C03645=1217.318,-29.503,-40.529,-179.892,5.418,148.913
C03646=1217.324,-29.753,-40.516,-179.895,5.418,148.914
C03647=1217.328,-30.003,-40.503,-179.897,5.418,148.915
C03648=1217.333,-30.252,-40.490,-179.899,5.417,148.915
C03649=1217.339,-30.503,-40.476,-179.902,5.417,148.916
C03650=1217.344,-30.752,-40.464,-179.904,5.417,148.917
C03651=1217.349,-31.001,-40.451,-179.907,5.417,148.918
C03652=1217.354,-31.252,-40.438,-179.909,5.416,148.918
C03653=1217.359,-31.501,-40.425,-179.912,5.417,148.919
C03654=1217.364,-31.750,-40.413,-179.914,5.416,148.920
C03655=1217.369,-32.000,-40.398,-179.917,5.416,148.920
C03656=1217.374,-32.249,-40.386,-179.919,5.416,148.921
C03657=1217.380,-32.499,-40.373,-179.922,5.415,148.922
C03658=1217.384,-32.749,-40.360,-179.924,5.415,148.922
C03659=1217.390,-32.998,-40.347,-179.926,5.415,148.923
C03660=1217.395,-33.248,-40.334,-179.928,5.414,148.924
C03661=1217.400,-33.498,-40.321,-179.931,5.414,148.924
C03662=1217.405,-33.747,-40.308,-179.933,5.414,148.925
C03663=1217.411,-33.997,-40.296,-179.936,5.414,148.926
C03664=1217.415,-34.247,-40.283,-179.939,5.413,148.926
C03665=1217.420,-34.496,-40.270,-179.941,5.414,148.927
C03666=1217.425,-34.745,-40.257,-179.943,5.413,148.928
C03667=1217.431,-34.996,-40.244,-179.946,5.413,148.928
C03668=1217.436,-35.245,-40.231,-179.948,5.413,148.929
C03669=1217.441,-35.494,-40.219,-179.951,5.412,148.930
C03670=1217.446,-35.743,-40.206,-179.953,5.412,148.931
C03671=1217.451,-35.994,-40.192,-179.955,5.412,148.931
C03672=1217.457,-36.244,-40.181,-179.958,5.412,148.932
C03673=1217.462,-36.493,-40.168,-179.961,5.411,148.933
C03674=1217.466,-36.743,-40.155,-179.963,5.412,148.933
C03675=1217.471,-36.992,-40.142,-179.966,5.411,148.934
C03676=1217.477,-37.242,-40.129,-179.968,5.411,148.935
C03677=1217.482,-37.491,-40.117,-179.970,5.411,148.935
C03678=1217.487,-37.741,-40.104,-179.973,5.411,148.936
C03679=1217.492,-37.991,-40.091,-179.975,5.411,148.937
C03680=1217.497,-38.240,-40.078,-179.978,5.410,148.938
C03681=1217.502,-38.489,-40.066,-179.980,5.410,148.938
C03682=1217.508,-38.740,-40.053,-179.982,5.410,148.939
C03683=1217.513,-38.990,-40.040,-179.985,5.409,148.939
C03684=1217.518,-39.239,-40.028,-179.987,5.409,148.940
C03685=1217.523,-39.488,-40.015,-179.989,5.409,148.941
C03686=1217.528,-39.738,-40.002,-179.992,5.409,148.942
C03687=1217.533,-39.988,-39.990,-179.995,5.408,148.942
C03688=1217.538,-40.238,-39.978,-179.997,5.409,148.943
C03689=1217.543,-40.487,-39.965,-179.999,5.408,148.944
C03690=1217.549,-40.737,-39.952,179.998,5.408,148.944
C03691=1217.554,-40.986,-39.939,179.996,5.408,148.945
C03692=1217.559,-41.236,-39.926,179.993,5.408,148.946
C03693=1217.564,-41.486,-39.914,179.991,5.407,148.946
C03694=1217.570,-41.735,-39.902,179.988,5.407,148.947
C03695=1217.574,-41.985,-39.889,179.986,5.407,148.948
C03696=1217.579,-42.234,-39.876,179.984,5.407,148.949
C03697=1217.585,-42.484,-39.864,179.981,5.407,148.949
C03698=1217.590,-42.734,-39.852,179.978,5.406,148.950
C03699=1217.595,-42.983,-39.839,179.976,5.407,148.951
C03700=1217.599,-43.233,-39.826,179.974,5.406,148.951
C03701=1217.605,-43.483,-39.814,179.971,5.406,148.952
C03702=1217.610,-43.732,-39.802,179.969,5.406,148.953
C03703=1217.615,-43.982,-39.789,179.967,5.405,148.953
C03704=1217.620,-44.231,-39.777,179.964,5.405,148.954
C03705=1217.625,-44.482,-39.764,179.962,5.405,148.955
C03706=1217.630,-44.731,-39.752,179.959,5.405,148.955
C03707=1217.635,-44.980,-39.739,179.957,5.405,148.956
C03708=1217.641,-45.230,-39.727,179.955,5.404,148.957
C03709=1217.646,-45.479,-39.715,179.952,5.404,148.957
C03710=1217.651,-45.729,-39.702,179.950,5.404,148.958
C03711=1217.656,-45.979,-39.690,179.947,5.404,148.959
C03712=1217.661,-46.229,-39.677,179.944,5.403,148.960
C03713=1217.666,-46.478,-39.665,179.942,5.404,148.960
C03714=1217.671,-46.728,-39.653,179.940,5.403,148.961
C03715=1217.677,-46.977,-39.640,179.938,5.404,148.962
C03716=1217.682,-47.227,-39.628,179.935,5.403,148.962
C03717=1217.687,-47.476,-39.616,179.932,5.403,148.963
C03718=1217.692,-47.726,-39.603,179.930,5.403,148.964
C03719=1217.697,-47.976,-39.591,179.928,5.402,148.964
C03720=1217.702,-48.226,-39.578,179.925,5.402,148.965
C03721=1217.708,-48.495,-39.566,179.923,5.402,148.966
C03722=1217.714,-48.765,-39.551,179.920,5.402,148.967
C03723=1217.719,-49.036,-39.538,179.917,5.401,148.967
C03724=1217.725,-49.305,-39.525,179.915,5.401,148.968
C03725=1217.730,-49.555,-39.513,179.913,5.401,148.969
C03726=1217.735,-49.805,-39.500,179.910,5.401,148.969
C03727=1217.740,-50.055,-39.488,179.908,5.401,148.970
C03728=1217.745,-50.304,-39.476,179.905,5.401,148.971
C03729=1217.751,-50.554,-39.464,179.903,5.400,148.971
C03730=1217.756,-50.803,-39.451,179.901,5.400,148.972
C03731=1217.760,-51.053,-39.440,179.898,5.400,148.973
C03732=1217.766,-51.302,-39.427,179.896,5.400,148.974
C03733=1217.771,-51.552,-39.415,179.893,5.400,148.974
C03734=1217.776,-51.801,-39.403,179.890,5.399,148.975
C03735=1217.782,-52.051,-39.391,179.888,5.400,148.976
C03736=1217.787,-52.301,-39.378,179.886,5.399,148.976
C03737=1217.792,-52.551,-39.366,179.883,5.399,148.977
C03738=1217.798,-52.801,-39.355,179.881,5.399,148.978
C03739=1217.801,-53.050,-39.342,179.878,5.399,148.979
C03740=1217.807,-53.300,-39.330,179.876,5.399,148.979
C03741=1217.812,-53.550,-39.318,179.874,5.399,148.980
C03742=1217.817,-53.800,-39.306,179.871,5.398,148.980
C03743=1217.822,-54.049,-39.293,179.869,5.398,148.981
C03744=1217.827,-54.298,-39.282,179.867,5.398,148.982
C03745=1217.833,-54.548,-39.270,179.865,5.398,148.982
C03746=1217.838,-54.798,-39.257,179.862,5.397,148.983
C03747=1217.843,-55.048,-39.245,179.859,5.397,148.984
C03748=1217.848,-55.297,-39.233,179.857,5.397,148.985
C03749=1217.853,-55.547,-39.222,179.854,5.397,148.985
C03750=1217.858,-55.797,-39.210,179.852,5.397,148.986
C03751=1217.863,-56.046,-39.197,179.850,5.397,148.987
C03752=1217.869,-56.296,-39.185,179.847,5.396,148.987
C03753=1217.874,-56.546,-39.173,179.845,5.397,148.988
C03754=1217.879,-56.795,-39.161,179.842,5.396,148.989
C03755=1217.884,-57.045,-39.149,179.840,5.397,148.990
C03756=1217.890,-57.295,-39.138,179.837,5.396,148.990
C03757=1217.895,-57.544,-39.125,179.835,5.396,148.991
C03758=1217.899,-57.794,-39.114,179.833,5.396,148.992
C03759=1217.905,-58.043,-39.102,179.830,5.395,148.992
C03760=1217.910,-58.293,-39.089,179.828,5.395,148.993
C03761=1217.915,-58.542,-39.078,179.826,5.395,148.994
C03762=1217.920,-58.792,-39.066,179.824,5.395,148.994
C03763=1217.926,-59.042,-39.054,179.821,5.395,148.995
C03764=1217.931,-59.292,-39.042,179.818,5.394,148.996
C03765=1217.935,-59.541,-39.030,179.816,5.395,148.996
C03766=1217.941,-59.791,-39.018,179.814,5.394,148.997
C03767=1217.946,-60.040,-39.006,179.812,5.395,148.998
C03768=1217.951,-60.290,-38.994,179.809,5.394,148.998
C03769=1217.956,-60.540,-38.983,179.806,5.394,148.999
C03770=1217.961,-60.790,-38.971,179.804,5.394,149.000
C03771=1217.966,-61.040,-38.959,179.801,5.394,149.001
C03772=1217.971,-61.289,-38.947,179.799,5.394,149.001
C03773=1217.977,-61.539,-38.935,179.797,5.393,149.002
C03774=1217.982,-61.788,-38.924,179.795,5.394,149.003
C03775=1217.987,-62.038,-38.912,179.792,5.393,149.003
C03776=1217.993,-62.288,-38.900,179.790,5.393,149.004
C03777=1217.997,-62.537,-38.888,179.788,5.393,149.005
C03778=1218.003,-62.787,-38.876,179.785,5.392,149.005
C03779=1218.008,-63.037,-38.864,179.783,5.393,149.006
C03780=1218.013,-63.286,-38.853,179.780,5.392,149.007
C03781=1218.018,-63.536,-38.841,179.778,5.392,149.007
C03782=1218.024,-63.786,-38.829,179.776,5.392,149.008
C03783=1218.028,-64.036,-38.818,179.773,5.392,149.009
C03784=1218.033,-64.285,-38.806,179.771,5.392,149.010
C03785=1218.038,-64.535,-38.794,179.768,5.392,149.010
C03786=1218.044,-64.784,-38.783,179.766,5.392,149.011
C03787=1218.050,-65.034,-38.771,179.763,5.391,149.012
C03788=1218.054,-65.283,-38.760,179.761,5.391,149.012
C03789=1218.060,-65.533,-38.748,179.759,5.391,149.013
C03790=1218.064,-65.783,-38.736,179.756,5.391,149.014
C03791=1218.070,-66.033,-38.724,179.754,5.391,149.014
C03792=1218.075,-66.283,-38.713,179.752,5.390,149.015
C03793=1218.080,-66.532,-38.701,179.750,5.391,149.016
C03794=1218.086,-66.782,-38.690,179.747,5.390,149.016
C03795=1218.091,-67.031,-38.678,179.744,5.390,149.017
C03796=1218.096,-67.281,-38.667,179.742,5.390,149.018
C03797=1218.101,-67.531,-38.655,179.739,5.390,149.018
C03798=1218.106,-67.780,-38.643,179.737,5.390,149.019
C03799=1218.111,-68.030,-38.631,179.735,5.390,149.020
C03800=1218.116,-68.280,-38.620,179.733,5.390,149.021
C03801=1218.122,-68.529,-38.608,179.730,5.390,149.021
C03802=1218.127,-68.779,-38.597,179.728,5.390,149.022
C03803=1218.132,-69.029,-38.585,179.725,5.389,149.023
C03804=1218.137,-69.279,-38.574,179.723,5.389,149.023
C03805=1218.143,-69.529,-38.562,179.720,5.389,149.024
C03806=1218.147,-69.778,-38.551,179.718,5.389,149.025
C03807=1218.153,-70.028,-38.540,179.716,5.389,149.025
C03808=1218.158,-70.277,-38.528,179.714,5.388,149.026
C03809=1218.163,-70.527,-38.516,179.711,5.389,149.027
C03810=1218.168,-70.777,-38.505,179.709,5.388,149.027
C03811=1218.174,-71.027,-38.493,179.706,5.388,149.028
C03812=1218.179,-71.276,-38.482,179.704,5.388,149.029
C03813=1218.184,-71.526,-38.470,179.701,5.388,149.030
C03814=1218.189,-71.775,-38.459,179.699,5.388,149.030
C03815=1218.194,-72.025,-38.448,179.697,5.388,149.031
C03816=1218.199,-72.275,-38.436,179.694,5.388,149.032
C03817=1218.204,-72.524,-38.425,179.692,5.388,149.032
C03818=1218.210,-72.774,-38.414,179.690,5.388,149.033
C03819=1218.215,-73.024,-38.403,179.688,5.387,149.034
C03820=1218.220,-73.274,-38.391,179.685,5.387,149.034
C03821=1218.226,-73.523,-38.380,179.683,5.387,149.035
C03822=1218.231,-73.773,-38.368,179.680,5.387,149.036
C03823=1218.236,-74.022,-38.357,179.678,5.387,149.036
C03824=1218.240,-74.272,-38.345,179.675,5.386,149.037
C03825=1218.247,-74.542,-38.333,179.673,5.387,149.038
C03826=1218.252,-74.813,-38.321,179.671,5.386,149.039
C03827=1218.258,-75.084,-38.309,179.667,5.386,149.039
C03828=1218.264,-75.354,-38.296,179.665,5.387,149.040
C03829=1218.268,-75.603,-38.285,179.663,5.386,149.041
C03830=1218.274,-75.854,-38.274,179.660,5.386,149.042
C03831=1218.279,-76.103,-38.263,179.658,5.386,149.042
C03832=1218.284,-76.353,-38.252,179.656,5.385,149.043
C03833=1218.290,-76.603,-38.240,179.654,5.386,149.044
C03834=1218.295,-76.853,-38.229,179.651,5.385,149.044
C03835=1218.301,-77.102,-38.218,179.649,5.386,149.045
C03836=1218.305,-77.352,-38.206,179.646,5.385,149.046
C03837=1218.310,-77.601,-38.195,179.644,5.385,149.046
C03838=1218.316,-77.852,-38.184,179.641,5.385,149.047
C03839=1218.321,-78.101,-38.173,179.639,5.385,149.048
C03840=1218.326,-78.350,-38.162,179.637,5.385,149.048
C03841=1218.331,-78.600,-38.150,179.635,5.385,149.049
C03842=1218.337,-78.850,-38.140,179.632,5.384,149.050
C03843=1218.341,-79.099,-38.128,179.630,5.384,149.050
C03844=1218.346,-79.349,-38.117,179.628,5.384,149.051
C03845=1218.352,-79.599,-38.106,179.625,5.384,149.052
C03846=1218.357,-79.849,-38.095,179.623,5.384,149.052
C03847=1218.362,-80.098,-38.084,179.620,5.384,149.053
C03848=1218.368,-80.349,-38.072,179.618,5.384,149.054
C03849=1218.373,-80.598,-38.062,179.615,5.384,149.055
C03850=1218.378,-80.847,-38.050,179.613,5.384,149.055
C03851=1218.383,-81.098,-38.039,179.611,5.384,149.056
C03852=1218.389,-81.347,-38.028,179.609,5.384,149.057
C03853=1218.393,-81.596,-38.017,179.606,5.383,149.057
C03854=1218.398,-81.847,-38.006,179.604,5.384,149.058
C03855=1218.404,-82.096,-37.995,179.602,5.383,149.059
C03856=1218.409,-82.345,-37.983,179.600,5.383,149.059
C03857=1218.414,-82.596,-37.973,179.597,5.383,149.060
C03858=1218.419,-82.845,-37.962,179.594,5.383,149.061
C03859=1218.425,-83.095,-37.951,179.592,5.383,149.061
C03860=1218.430,-83.344,-37.940,179.589,5.382,149.062
C03861=1218.435,-83.594,-37.929,179.587,5.383,149.063
C03862=1218.440,-83.844,-37.918,179.585,5.382,149.064
C03863=1218.445,-84.093,-37.907,179.583,5.382,149.064
C03864=1218.451,-84.343,-37.896,179.580,5.382,149.065
C03865=1218.456,-84.593,-37.885,179.578,5.382,149.066
C03866=1218.461,-84.843,-37.874,179.576,5.382,149.066
C03867=1218.466,-85.092,-37.863,179.574,5.382,149.067
C03868=1218.471,-85.343,-37.853,179.571,5.382,149.068
C03869=1218.477,-85.592,-37.841,179.569,5.382,149.068
C03870=1218.482,-85.842,-37.830,179.566,5.382,149.069
C03871=1218.487,-86.091,-37.820,179.564,5.382,149.070
C03872=1218.492,-86.341,-37.809,179.562,5.381,149.070
C03873=1218.497,-86.591,-37.798,179.560,5.382,149.071
C03874=1218.503,-86.840,-37.787,179.557,5.381,149.072
C03875=1218.508,-87.090,-37.776,179.555,5.382,149.072
C03876=1218.514,-87.340,-37.765,179.552,5.381,149.073
C03877=1218.518,-87.589,-37.754,179.550,5.381,149.074
C03878=1218.523,-87.840,-37.743,179.548,5.381,149.075
C03879=1218.529,-88.089,-37.733,179.545,5.381,149.075
C03880=1218.534,-88.339,-37.722,179.543,5.381,149.076
C03881=1218.539,-88.588,-37.711,179.540,5.380,149.077
C03882=1218.544,-88.838,-37.700,179.539,5.380,149.077
C03883=1218.550,-89.087,-37.689,179.536,5.380,149.078
C03884=1218.555,-89.338,-37.678,179.534,5.380,149.079
C03885=1218.560,-89.588,-37.668,179.531,5.380,149.079
C03886=1218.565,-89.837,-37.657,179.529,5.380,149.080
C03887=1218.570,-90.087,-37.646,179.526,5.380,149.081
C03888=1218.576,-90.336,-37.635,179.524,5.380,149.081
C03889=1218.581,-90.586,-37.625,179.522,5.380,149.082
C03890=1218.586,-90.836,-37.615,179.520,5.380,149.083
C03891=1218.591,-91.085,-37.603,179.517,5.379,149.083
C03892=1218.596,-91.335,-37.593,179.515,5.380,149.084
C03893=1218.601,-91.585,-37.583,179.513,5.379,149.085
C03894=1218.607,-91.834,-37.571,179.510,5.380,149.085
C03895=1218.612,-92.085,-37.560,179.508,5.379,149.086
C03896=1218.618,-92.333,-37.550,179.506,5.380,149.087
C03897=1218.623,-92.584,-37.539,179.503,5.379,149.088
C03898=1218.628,-92.834,-37.528,179.501,5.379,149.088
C03899=1218.633,-93.083,-37.518,179.499,5.379,149.089
C03900=1218.638,-93.333,-37.507,179.497,5.379,149.089
C03901=1218.644,-93.583,-37.497,179.494,5.379,149.090
C03902=1218.649,-93.833,-37.486,179.492,5.379,149.091
C03903=1218.654,-94.082,-37.475,179.489,5.379,149.092
C03904=1218.659,-94.332,-37.465,179.487,5.379,149.092
C03905=1218.665,-94.582,-37.454,179.484,5.378,149.093
C03906=1218.669,-94.831,-37.443,179.483,5.378,149.094
C03907=1218.675,-95.081,-37.433,179.480,5.378,149.094
C03908=1218.680,-95.330,-37.423,179.478,5.378,149.095
C03909=1218.685,-95.581,-37.412,179.475,5.378,149.096
C03910=1218.691,-95.829,-37.401,179.473,5.378,149.096
C03911=1218.696,-96.080,-37.391,179.471,5.378,149.097
C03912=1218.701,-96.329,-37.380,179.469,5.378,149.098
C03913=1218.706,-96.580,-37.370,179.466,5.378,149.099
C03914=1218.712,-96.829,-37.360,179.464,5.378,149.099
C03915=1218.717,-97.079,-37.348,179.462,5.377,149.100
C03916=1218.722,-97.328,-37.338,179.460,5.378,149.100
C03917=1218.727,-97.578,-37.328,179.457,5.377,149.101
C03918=1218.733,-97.828,-37.317,179.455,5.378,149.102
C03919=1218.738,-98.078,-37.307,179.452,5.377,149.103
C03920=1218.742,-98.327,-37.296,179.450,5.378,149.103
C03921=1218.748,-98.576,-37.286,179.448,5.377,149.104
C03922=1218.753,-98.827,-37.276,179.446,5.377,149.104
C03923=1218.759,-99.076,-37.265,179.443,5.377,149.105
C03924=1218.764,-99.326,-37.255,179.441,5.377,149.106
C03925=1218.769,-99.576,-37.245,179.438,5.377,149.107
C03926=1218.774,-99.826,-37.234,179.436,5.377,149.107
C03927=1218.779,-100.075,-37.223,179.434,5.377,149.108
C03928=1218.785,-100.325,-37.213,179.432,5.377,149.109
C03929=1218.790,-100.596,-37.202,179.429,5.377,149.109
C03930=1218.796,-100.868,-37.190,179.427,5.377,149.110
C03931=1218.801,-101.139,-37.180,179.424,5.377,149.111
C03932=1218.808,-101.410,-37.168,179.421,5.376,149.112
C03933=1218.813,-101.659,-37.157,179.419,5.376,149.112
C03934=1218.817,-101.909,-37.147,179.417,5.376,149.113
C03935=1218.823,-102.158,-37.137,179.415,5.376,149.114
C03936=1218.828,-102.408,-37.127,179.412,5.376,149.114
C03937=1218.834,-102.658,-37.116,179.410,5.376,149.115
C03938=1218.839,-102.908,-37.106,179.407,5.376,149.116
C03939=1218.844,-103.158,-37.096,179.405,5.376,149.116
C03940=1218.849,-103.407,-37.086,179.403,5.376,149.117
C03941=1218.854,-103.657,-37.076,179.401,5.376,149.118
C03942=1218.860,-103.907,-37.065,179.398,5.375,149.118
C03943=1218.865,-104.157,-37.055,179.396,5.375,149.119
C03944=1218.870,-104.407,-37.045,179.394,5.375,149.120
C03945=1218.876,-104.656,-37.034,179.392,5.375,149.120
C03946=1218.880,-104.906,-37.024,179.389,5.375,149.121
C03947=1218.886,-105.156,-37.014,179.387,5.375,149.122
C03948=1218.891,-105.405,-37.004,179.385,5.375,149.122
C03949=1218.896,-105.655,-36.993,179.383,5.375,149.123
C03950=1218.902,-105.905,-36.983,179.380,5.375,149.124
C03951=1218.907,-106.154,-36.974,179.378,5.375,149.124
C03952=1218.912,-106.404,-36.963,179.376,5.375,149.125
C03953=1218.917,-106.654,-36.953,179.373,5.375,149.126
C03954=1218.923,-106.904,-36.943,179.371,5.375,149.126
C03955=1218.927,-107.153,-36.933,179.369,5.374,149.127
C03956=1218.933,-107.403,-36.922,179.367,5.375,149.128
C03957=1218.938,-107.653,-36.912,179.364,5.374,149.129
C03958=1218.944,-107.903,-36.902,179.362,5.375,149.129
C03959=1218.949,-108.153,-36.893,179.359,5.374,149.130
C03960=1218.954,-108.402,-36.882,179.358,5.374,149.130
C03961=1218.959,-108.652,-36.872,179.355,5.374,149.131
C03962=1218.965,-108.902,-36.862,179.353,5.374,149.132
C03963=1218.970,-109.151,-36.852,179.350,5.374,149.133
C03964=1218.975,-109.401,-36.841,179.348,5.374,149.133
C03965=1218.980,-109.651,-36.831,179.346,5.373,149.134
C03966=1218.985,-109.900,-36.822,179.344,5.374,149.135
C03967=1218.991,-110.150,-36.812,179.341,5.373,149.135
C03968=1218.996,-110.401,-36.802,179.339,5.374,149.136
C03969=1219.002,-110.650,-36.791,179.336,5.373,149.137
C03970=1219.006,-110.899,-36.782,179.334,5.374,149.137
C03971=1219.011,-111.150,-36.771,179.333,5.374,149.138
C03972=1219.017,-111.399,-36.761,179.330,5.373,149.139
C03973=1219.022,-111.649,-36.752,179.328,5.374,149.139
C03974=1219.028,-111.899,-36.742,179.325,5.373,149.140
C03975=1219.033,-112.149,-36.731,179.323,5.374,149.141
C03976=1219.038,-112.398,-36.722,179.321,5.373,149.141
C03977=1219.043,-112.648,-36.711,179.319,5.373,149.142
C03978=1219.049,-112.898,-36.702,179.316,5.373,149.143
C03979=1219.053,-113.148,-36.692,179.314,5.373,149.143
C03980=1219.059,-113.397,-36.682,179.311,5.373,149.144
C03981=1219.065,-113.647,-36.672,179.309,5.373,149.145
C03982=1219.070,-113.897,-36.663,179.307,5.372,149.145
C03983=1219.075,-114.147,-36.652,179.305,5.373,149.146
C03984=1219.080,-114.396,-36.642,179.302,5.372,149.147
C03985=1219.085,-114.646,-36.632,179.300,5.373,149.147
C03986=1219.091,-114.896,-36.623,179.298,5.372,149.148
C03987=1219.096,-115.145,-36.613,179.296,5.372,149.149
C03988=1219.101,-115.395,-36.603,179.294,5.373,149.149
C03989=1219.106,-115.645,-36.593,179.291,5.372,149.150
C03990=1219.112,-115.895,-36.583,179.289,5.373,149.151
C03991=1219.117,-116.144,-36.573,179.286,5.372,149.151
C03992=1219.122,-116.393,-36.564,179.285,5.372,149.152
C03993=1219.128,-116.644,-36.554,179.282,5.372,149.153
C03994=1219.132,-116.894,-36.544,179.280,5.372,149.153
C03995=1219.138,-117.143,-36.534,179.277,5.372,149.154
C03996=1219.144,-117.393,-36.524,179.275,5.372,149.155
C03997=1219.149,-117.642,-36.515,179.273,5.371,149.155
C03998=1219.154,-117.893,-36.504,179.271,5.372,149.156
C03999=1219.159,-118.143,-36.495,179.268,5.371,149.157
C04000=1219.164,-118.392,-36.485,179.266,5.372,149.157
C04001=1219.169,-118.641,-36.476,179.264,5.372,149.158
C04002=1219.175,-118.892,-36.466,179.262,5.371,149.159
C04003=1219.180,-119.141,-36.456,179.260,5.372,149.159
C04004=1219.185,-119.392,-36.447,179.257,5.371,149.160
C04005=1219.190,-119.641,-36.437,179.255,5.372,149.161
C04006=1219.196,-119.890,-36.427,179.253,5.371,149.161
C04007=1219.201,-120.140,-36.418,179.251,5.371,149.162
C04008=1219.207,-120.390,-36.408,179.248,5.371,149.163
C04009=1219.211,-120.640,-36.398,179.246,5.371,149.163
C04010=1219.217,-120.890,-36.388,179.243,5.371,149.164
C04011=1219.222,-121.139,-36.379,179.242,5.371,149.165
C04012=1219.228,-121.389,-36.369,179.239,5.370,149.165
C04013=1219.232,-121.639,-36.360,179.237,5.371,149.166
C04014=1219.238,-121.889,-36.350,179.235,5.371,149.167
C04015=1219.243,-122.138,-36.340,179.233,5.370,149.167
C04016=1219.248,-122.389,-36.331,179.231,5.371,149.168
C04017=1219.253,-122.638,-36.321,179.228,5.370,149.169
C04018=1219.259,-122.888,-36.311,179.226,5.371,149.169
C04019=1219.264,-123.137,-36.302,179.223,5.370,149.170
C04020=1219.270,-123.388,-36.292,179.222,5.370,149.171
C04021=1219.275,-123.637,-36.283,179.219,5.370,149.171
C04022=1219.280,-123.887,-36.274,179.217,5.370,149.172
C04023=1219.286,-124.136,-36.264,179.214,5.370,149.173
C04024=1219.290,-124.387,-36.254,179.212,5.370,149.173
C04025=1219.296,-124.636,-36.244,179.210,5.370,149.174
C04026=1219.301,-124.886,-36.235,179.208,5.370,149.175
C04027=1219.307,-125.136,-36.225,179.206,5.370,149.175
C04028=1219.312,-125.386,-36.216,179.203,5.369,149.176
C04029=1219.317,-125.635,-36.207,179.201,5.370,149.177
C04030=1219.323,-125.885,-36.197,179.199,5.369,149.177
C04031=1219.328,-126.135,-36.188,179.197,5.370,149.178
C04032=1219.333,-126.384,-36.178,179.194,5.369,149.179
C04033=1218.912,-126.395,-36.214,179.190,5.372,149.181
C04034=1218.906,-126.146,-36.224,179.193,5.373,149.180
C04035=1218.901,-125.896,-36.233,179.195,5.372,149.179
C04036=1218.895,-125.646,-36.244,179.197,5.373,149.179
C04037=1218.890,-125.396,-36.252,179.199,5.373,149.178
C04038=1218.885,-125.147,-36.262,179.202,5.373,149.177
C04039=1218.880,-124.896,-36.272,179.204,5.373,149.177
C04040=1218.875,-124.647,-36.282,179.206,5.374,149.176
C04041=1218.869,-124.397,-36.291,179.208,5.373,149.175
C04042=1218.864,-124.147,-36.300,179.210,5.373,149.175
C04043=1218.858,-123.897,-36.310,179.213,5.373,149.174
C04044=1218.853,-123.648,-36.319,179.214,5.373,149.173
C04045=1218.848,-123.398,-36.329,179.217,5.374,149.173
C04046=1218.842,-123.148,-36.338,179.219,5.373,149.172
C04047=1218.838,-122.899,-36.348,179.222,5.374,149.171
C04048=1218.832,-122.649,-36.357,179.223,5.374,149.171
C04049=1218.827,-122.399,-36.367,179.226,5.374,149.170
C04050=1218.821,-122.149,-36.377,179.228,5.374,149.169
C04051=1218.817,-121.899,-36.386,179.231,5.374,149.169
C04052=1218.811,-121.650,-36.397,179.233,5.374,149.168
C04053=1218.806,-121.400,-36.405,179.235,5.374,149.167
C04054=1218.800,-121.150,-36.416,179.237,5.374,149.167
C04055=1218.795,-120.901,-36.425,179.239,5.374,149.166
C04056=1218.790,-120.650,-36.435,179.242,5.374,149.165
C04057=1218.785,-120.401,-36.444,179.244,5.374,149.165
C04058=1218.779,-120.151,-36.454,179.246,5.375,149.164
C04059=1218.774,-119.902,-36.464,179.248,5.374,149.163
C04060=1218.769,-119.652,-36.473,179.251,5.375,149.163
C04061=1218.764,-119.402,-36.483,179.253,5.374,149.162
C04062=1218.758,-119.152,-36.493,179.255,5.375,149.161
C04063=1218.753,-118.902,-36.502,179.257,5.375,149.161
C04064=1218.748,-118.653,-36.513,179.260,5.375,149.160
C04065=1218.743,-118.403,-36.522,179.262,5.375,149.159
C04066=1218.737,-118.153,-36.532,179.264,5.375,149.159
C04067=1218.732,-117.903,-36.541,179.267,5.375,149.158
C04068=1218.727,-117.653,-36.551,179.269,5.375,149.157
C04069=1218.722,-117.404,-36.561,179.271,5.375,149.157
C04070=1218.716,-117.154,-36.570,179.273,5.375,149.156
C04071=1218.711,-116.905,-36.580,179.276,5.376,149.155
C04072=1218.706,-116.655,-36.590,179.278,5.375,149.155
C04073=1218.700,-116.404,-36.600,179.280,5.376,149.154
C04074=1218.696,-116.155,-36.610,179.282,5.375,149.153
C04075=1218.690,-115.905,-36.620,179.285,5.376,149.153
C04076=1218.685,-115.656,-36.629,179.287,5.376,149.152
C04077=1218.679,-115.406,-36.639,179.289,5.376,149.151
C04078=1218.674,-115.156,-36.650,179.292,5.376,149.151
C04079=1218.669,-114.907,-36.659,179.294,5.375,149.150
C04080=1218.663,-114.656,-36.669,179.296,5.376,149.149
C04081=1218.659,-114.407,-36.678,179.298,5.376,149.149
C04082=1218.654,-114.157,-36.689,179.301,5.376,149.148
C04083=1218.648,-113.907,-36.699,179.303,5.376,149.147
C04084=1218.643,-113.658,-36.708,179.305,5.376,149.147
C04085=1218.637,-113.408,-36.718,179.307,5.376,149.146
C04086=1218.632,-113.158,-36.728,179.310,5.377,149.145
C04087=1218.627,-112.909,-36.738,179.312,5.376,149.145
C04088=1218.621,-112.658,-36.748,179.314,5.377,149.144
C04089=1218.616,-112.409,-36.758,179.316,5.376,149.143
C04090=1218.611,-112.160,-36.768,179.319,5.377,149.143
C04091=1218.606,-111.909,-36.778,179.321,5.377,149.142
C04092=1218.600,-111.660,-36.788,179.323,5.377,149.141
C04093=1218.595,-111.410,-36.797,179.326,5.377,149.141
C04094=1218.590,-111.160,-36.808,179.328,5.377,149.140
C04095=1218.585,-110.910,-36.818,179.330,5.377,149.139
C04096=1218.580,-110.661,-36.828,179.332,5.376,149.139
C04097=1218.574,-110.411,-36.838,179.335,5.377,149.138
C04098=1218.569,-110.160,-36.848,179.337,5.377,149.137
C04099=1218.564,-109.911,-36.857,179.339,5.377,149.137
C04100=1218.558,-109.662,-36.868,179.341,5.377,149.136
C04101=1218.553,-109.412,-36.878,179.344,5.377,149.135
C04102=1218.549,-109.162,-36.888,179.346,5.377,149.135
C04103=1218.543,-108.913,-36.898,179.348,5.378,149.134
C04104=1218.537,-108.663,-36.908,179.350,5.377,149.133
C04105=1218.532,-108.413,-36.919,179.353,5.378,149.133
C04106=1218.527,-108.163,-36.928,179.355,5.377,149.132
C04107=1218.522,-107.914,-36.938,179.358,5.378,149.131
C04108=1218.517,-107.663,-36.948,179.360,5.378,149.131
C04109=1218.511,-107.414,-36.959,179.362,5.378,149.130
C04110=1218.506,-107.165,-36.968,179.364,5.378,149.129
C04111=1218.501,-106.914,-36.979,179.367,5.378,149.128
C04112=1218.496,-106.665,-36.989,179.369,5.378,149.128
C04113=1218.490,-106.415,-36.999,179.372,5.378,149.127
C04114=1218.486,-106.165,-37.009,179.373,5.378,149.127
C04115=1218.480,-105.916,-37.019,179.376,5.379,149.126
C04116=1218.475,-105.666,-37.030,179.378,5.378,149.125
C04117=1218.470,-105.416,-37.040,179.381,5.379,149.124
C04118=1218.464,-105.166,-37.050,179.383,5.378,149.124
C04119=1218.459,-104.917,-37.060,179.385,5.378,149.123
C04120=1218.454,-104.667,-37.071,179.387,5.379,149.123
C04121=1218.448,-104.417,-37.081,179.389,5.379,149.122
C04122=1218.443,-104.168,-37.091,179.392,5.379,149.121
C04123=1218.438,-103.918,-37.102,179.394,5.379,149.120
C04124=1218.433,-103.668,-37.111,179.397,5.379,149.120
C04125=1218.428,-103.418,-37.122,179.399,5.379,149.119
C04126=1218.422,-103.169,-37.132,179.401,5.379,149.118
C04127=1218.417,-102.919,-37.142,179.403,5.379,149.118
C04128=1218.412,-102.669,-37.153,179.406,5.380,149.117
C04129=1218.406,-102.419,-37.163,179.408,5.379,149.116
C04130=1218.401,-102.170,-37.173,179.410,5.380,149.116
C04131=1218.396,-101.920,-37.183,179.413,5.379,149.115
C04132=1218.391,-101.670,-37.193,179.415,5.380,149.114
C04133=1218.386,-101.420,-37.204,179.417,5.380,149.114
C04134=1218.380,-101.149,-37.215,179.420,5.380,149.113
C04135=1218.374,-100.878,-37.227,179.423,5.380,149.112
C04136=1218.369,-100.607,-37.238,179.425,5.380,149.111
C04137=1218.363,-100.336,-37.249,179.427,5.380,149.111
C04138=1218.358,-100.086,-37.260,179.430,5.380,149.110
C04139=1218.352,-99.836,-37.270,179.432,5.381,149.109
C04140=1218.347,-99.586,-37.280,179.434,5.380,149.109
C04141=1218.342,-99.337,-37.290,179.437,5.381,149.108
C04142=1218.337,-99.087,-37.301,179.439,5.380,149.107
C04143=1218.332,-98.838,-37.311,179.441,5.381,149.107
C04144=1218.326,-98.588,-37.322,179.443,5.380,149.106
C04145=1218.321,-98.338,-37.332,179.446,5.381,149.105
C04146=1218.316,-98.088,-37.342,179.448,5.381,149.105
C04147=1218.311,-97.838,-37.353,179.450,5.381,149.104
C04148=1218.305,-97.589,-37.364,179.452,5.381,149.103
C04149=1218.300,-97.339,-37.374,179.455,5.381,149.103
C04150=1218.295,-97.089,-37.385,179.457,5.381,149.102
C04151=1218.290,-96.839,-37.395,179.460,5.381,149.101
C04152=1218.284,-96.590,-37.405,179.462,5.381,149.100
C04153=1218.279,-96.341,-37.416,179.464,5.382,149.100
C04154=1218.274,-96.090,-37.427,179.466,5.381,149.099
C04155=1218.268,-95.841,-37.437,179.469,5.382,149.098
C04156=1218.263,-95.591,-37.448,179.471,5.381,149.098
C04157=1218.258,-95.341,-37.458,179.474,5.382,149.097
C04158=1218.253,-95.092,-37.469,179.476,5.382,149.096
C04159=1218.247,-94.842,-37.479,179.478,5.382,149.096
C04160=1218.242,-94.592,-37.490,179.480,5.382,149.095
C04161=1218.237,-94.342,-37.500,179.483,5.382,149.094
C04162=1218.232,-94.093,-37.512,179.485,5.382,149.094
C04163=1218.227,-93.843,-37.522,179.487,5.382,149.093
C04164=1218.222,-93.593,-37.532,179.490,5.382,149.092
C04165=1218.216,-93.344,-37.543,179.492,5.383,149.092
C04166=1218.211,-93.094,-37.554,179.494,5.382,149.091
C04167=1218.206,-92.844,-37.564,179.497,5.383,149.090
C04168=1218.201,-92.594,-37.575,179.499,5.383,149.090
C04169=1218.195,-92.345,-37.586,179.501,5.383,149.089
C04170=1218.190,-92.095,-37.596,179.503,5.383,149.088
C04171=1218.185,-91.846,-37.607,179.506,5.383,149.088
C04172=1218.180,-91.595,-37.618,179.508,5.383,149.087
C04173=1218.174,-91.346,-37.628,179.511,5.383,149.086
C04174=1218.170,-91.096,-37.639,179.513,5.383,149.085
C04175=1218.164,-90.847,-37.649,179.516,5.383,149.085
C04176=1218.159,-90.597,-37.660,179.517,5.383,149.084
C04177=1218.155,-90.347,-37.671,179.520,5.384,149.084
C04178=1218.149,-90.097,-37.681,179.522,5.383,149.083
C04179=1218.143,-89.847,-37.693,179.525,5.384,149.082
C04180=1218.138,-89.598,-37.703,179.527,5.383,149.081
C04181=1218.133,-89.348,-37.714,179.529,5.384,149.081
C04182=1218.128,-89.099,-37.725,179.531,5.384,149.080
C04183=1218.123,-88.848,-37.736,179.534,5.384,149.079
C04184=1218.117,-88.600,-37.746,179.536,5.384,149.079
C04185=1218.112,-88.349,-37.757,179.538,5.384,149.078
C04186=1218.107,-88.099,-37.768,179.541,5.385,149.077
C04187=1218.102,-87.850,-37.779,179.543,5.384,149.077
C04188=1218.096,-87.600,-37.790,179.546,5.385,149.076
C04189=1218.091,-87.351,-37.801,179.548,5.385,149.075
C04190=1218.086,-87.100,-37.811,179.551,5.385,149.074
C04191=1218.081,-86.851,-37.823,179.553,5.385,149.074
C04192=1218.076,-86.601,-37.833,179.555,5.385,149.073
C04193=1218.071,-86.352,-37.844,179.557,5.385,149.073
C04194=1218.065,-86.102,-37.854,179.560,5.386,149.072
C04195=1218.060,-85.852,-37.866,179.562,5.385,149.071
C04196=1218.055,-85.602,-37.877,179.564,5.386,149.070
C04197=1218.050,-85.353,-37.888,179.566,5.385,149.070
C04198=1218.045,-85.103,-37.898,179.569,5.386,149.069
C04199=1218.039,-84.854,-37.909,179.571,5.385,149.068
C04200=1218.034,-84.603,-37.920,179.574,5.386,149.068
C04201=1218.029,-84.354,-37.932,179.576,5.385,149.067
C04202=1218.023,-84.104,-37.942,179.579,5.386,149.066
C04203=1218.019,-83.854,-37.953,179.580,5.386,149.066
C04204=1218.014,-83.605,-37.964,179.583,5.386,149.065
C04205=1218.008,-83.355,-37.975,179.585,5.386,149.064
C04206=1218.003,-83.105,-37.986,179.588,5.386,149.064
C04207=1217.997,-82.856,-37.997,179.590,5.387,149.063
C04208=1217.993,-82.606,-38.008,179.592,5.386,149.062
C04209=1217.988,-82.357,-38.019,179.595,5.387,149.061
C04210=1217.982,-82.107,-38.030,179.597,5.387,149.061
C04211=1217.977,-81.857,-38.041,179.600,5.387,149.060
C04212=1217.972,-81.607,-38.052,179.601,5.387,149.060
C04213=1217.967,-81.358,-38.063,179.604,5.387,149.059
C04214=1217.961,-81.108,-38.075,179.606,5.387,149.058
C04215=1217.956,-80.858,-38.085,179.609,5.388,149.057
C04216=1217.951,-80.609,-38.096,179.611,5.387,149.057
C04217=1217.946,-80.359,-38.108,179.614,5.388,149.056
C04218=1217.941,-80.109,-38.119,179.616,5.387,149.055
C04219=1217.935,-79.860,-38.130,179.618,5.388,149.055
C04220=1217.931,-79.610,-38.141,179.621,5.387,149.054
C04221=1217.925,-79.360,-38.152,179.623,5.388,149.053
C04222=1217.920,-79.110,-38.163,179.626,5.388,149.052
C04223=1217.915,-78.861,-38.174,179.627,5.388,149.052
C04224=1217.909,-78.610,-38.185,179.630,5.389,149.051
C04225=1217.904,-78.361,-38.197,179.632,5.388,149.051
C04226=1217.899,-78.112,-38.208,179.635,5.389,149.050
C04227=1217.894,-77.862,-38.220,179.637,5.388,149.049
C04228=1217.889,-77.612,-38.230,179.640,5.389,149.048
C04229=1217.884,-77.362,-38.241,179.642,5.389,149.048
C04230=1217.878,-77.113,-38.253,179.644,5.389,149.047
C04231=1217.873,-76.863,-38.263,179.647,5.389,149.046
C04232=1217.868,-76.613,-38.275,179.649,5.389,149.046
C04233=1217.862,-76.364,-38.286,179.651,5.389,149.045
C04234=1217.858,-76.114,-38.298,179.653,5.390,149.044
C04235=1217.852,-75.864,-38.309,179.656,5.390,149.044
C04236=1217.847,-75.614,-38.320,179.658,5.390,149.043
C04237=1217.842,-75.365,-38.331,179.661,5.390,149.042
C04238=1217.836,-75.094,-38.343,179.663,5.390,149.042
C04239=1217.831,-74.824,-38.356,179.666,5.390,149.041
C04240=1217.825,-74.553,-38.368,179.669,5.390,149.040
C04241=1217.819,-74.282,-38.380,179.671,5.390,149.039
C04242=1217.814,-74.033,-38.392,179.674,5.390,149.039
C04243=1217.808,-73.784,-38.403,179.676,5.390,149.038
C04244=1217.804,-73.534,-38.414,179.678,5.390,149.037
C04245=1217.799,-73.284,-38.426,179.681,5.391,149.037
C04246=1217.794,-73.034,-38.438,179.683,5.391,149.036
C04247=1217.788,-72.785,-38.448,179.685,5.391,149.035
C04248=1217.782,-72.535,-38.460,179.687,5.391,149.035
C04249=1217.778,-72.285,-38.471,179.690,5.391,149.034
C04250=1217.772,-72.035,-38.483,179.692,5.391,149.033
C04251=1217.768,-71.786,-38.494,179.695,5.392,149.032
C04252=1217.762,-71.536,-38.506,179.697,5.391,149.032
C04253=1217.757,-71.287,-38.517,179.700,5.392,149.031
C04254=1217.752,-71.037,-38.528,179.702,5.392,149.030
C04255=1217.747,-70.787,-38.540,179.704,5.392,149.030
C04256=1217.742,-70.538,-38.551,179.707,5.392,149.029
C04257=1217.736,-70.288,-38.562,179.709,5.392,149.028
C04258=1217.731,-70.038,-38.574,179.711,5.393,149.028
C04259=1217.726,-69.788,-38.585,179.713,5.392,149.027
C04260=1217.721,-69.539,-38.597,179.716,5.393,149.026
C04261=1217.716,-69.289,-38.609,179.719,5.393,149.026
C04262=1217.710,-69.040,-38.620,179.721,5.393,149.025
C04263=1217.705,-68.790,-38.631,179.723,5.393,149.024
C04264=1217.700,-68.540,-38.643,179.726,5.393,149.023
C04265=1217.695,-68.290,-38.655,179.728,5.393,149.023
C04266=1217.689,-68.040,-38.666,179.730,5.393,149.022
C04267=1217.685,-67.791,-38.678,179.733,5.394,149.021
C04268=1217.679,-67.541,-38.689,179.735,5.393,149.021
C04269=1217.674,-67.292,-38.701,179.738,5.394,149.020
C04270=1217.668,-67.042,-38.712,179.740,5.395,149.019
C04271=1217.664,-66.792,-38.724,179.742,5.394,149.019
C04272=1217.658,-66.542,-38.736,179.745,5.395,149.018
C04273=1217.654,-66.293,-38.747,179.747,5.394,149.017
C04274=1217.648,-66.043,-38.759,179.749,5.395,149.017
C04275=1217.642,-65.794,-38.771,179.751,5.394,149.016
C04276=1217.638,-65.544,-38.782,179.754,5.395,149.015
C04277=1217.632,-65.295,-38.794,179.757,5.395,149.014
C04278=1217.628,-65.045,-38.805,179.759,5.395,149.014
C04279=1217.622,-64.795,-38.817,179.762,5.395,149.013
C04280=1217.617,-64.545,-38.829,179.764,5.395,149.012
C04281=1217.612,-64.295,-38.841,179.766,5.396,149.012
C04282=1217.607,-64.045,-38.852,179.768,5.395,149.011
C04283=1217.602,-63.796,-38.864,179.771,5.396,149.010
C04284=1217.597,-63.546,-38.876,179.774,5.396,149.010
C04285=1217.591,-63.297,-38.888,179.775,5.396,149.009
C04286=1217.586,-63.048,-38.899,179.778,5.397,149.008
C04287=1217.581,-62.798,-38.911,179.780,5.396,149.008
C04288=1217.576,-62.548,-38.922,179.783,5.397,149.007
C04289=1217.571,-62.298,-38.934,179.785,5.397,149.006
C04290=1217.565,-62.048,-38.946,179.788,5.397,149.006
C04291=1217.561,-61.799,-38.958,179.790,5.397,149.005
C04292=1217.555,-61.549,-38.970,179.792,5.397,149.004
C04293=1217.550,-61.299,-38.982,179.795,5.397,149.003
C04294=1217.545,-61.050,-38.993,179.797,5.397,149.003
C04295=1217.540,-60.800,-39.005,179.800,5.397,149.002
C04296=1217.535,-60.550,-39.018,179.802,5.398,149.001
C04297=1217.530,-60.301,-39.029,179.804,5.398,149.001
C04298=1217.525,-60.051,-39.041,179.807,5.398,149.000
C04299=1217.519,-59.801,-39.053,179.809,5.398,148.999
C04300=1217.513,-59.552,-39.064,179.811,5.399,148.999
C04301=1217.509,-59.303,-39.076,179.814,5.399,148.998
C04302=1217.503,-59.053,-39.088,179.816,5.399,148.997
C04303=1217.498,-58.803,-39.100,179.819,5.399,148.997
C04304=1217.493,-58.554,-39.112,179.821,5.399,148.996
C04305=1217.488,-58.304,-39.124,179.824,5.399,148.995
C04306=1217.483,-58.054,-39.136,179.826,5.400,148.994
C04307=1217.477,-57.804,-39.148,179.828,5.399,148.994
C04308=1217.473,-57.555,-39.160,179.831,5.400,148.993
C04309=1217.467,-57.305,-39.172,179.833,5.399,148.992
C04310=1217.462,-57.055,-39.183,179.836,5.400,148.992
C04311=1217.457,-56.806,-39.196,179.838,5.400,148.991
C04312=1217.452,-56.556,-39.207,179.840,5.400,148.990
C04313=1217.447,-56.306,-39.219,179.843,5.401,148.990
C04314=1217.442,-56.057,-39.232,179.845,5.400,148.989
C04315=1217.436,-55.807,-39.244,179.848,5.401,148.988
C04316=1217.431,-55.557,-39.255,179.850,5.400,148.987
C04317=1217.426,-55.308,-39.268,179.852,5.401,148.987
C04318=1217.421,-55.058,-39.279,179.855,5.402,148.986
C04319=1217.416,-54.809,-39.292,179.857,5.401,148.986
C04320=1217.410,-54.559,-39.304,179.860,5.402,148.985
C04321=1217.406,-54.309,-39.316,179.862,5.401,148.984
C04322=1217.401,-54.059,-39.328,179.864,5.402,148.983
C04323=1217.396,-53.809,-39.340,179.867,5.402,148.983
C04324=1217.391,-53.560,-39.353,179.869,5.402,148.982
C04325=1217.385,-53.310,-39.365,179.872,5.402,148.981
C04326=1217.380,-53.060,-39.376,179.874,5.402,148.981
C04327=1217.375,-52.811,-39.388,179.876,5.403,148.980
C04328=1217.370,-52.561,-39.400,179.879,5.403,148.979
C04329=1217.365,-52.312,-39.413,179.881,5.403,148.978
C04330=1217.359,-52.062,-39.425,179.884,5.403,148.978
C04331=1217.354,-51.813,-39.437,179.887,5.404,148.977
C04332=1217.349,-51.563,-39.449,179.889,5.403,148.976
C04333=1217.344,-51.314,-39.461,179.891,5.404,148.976
C04334=1217.339,-51.064,-39.473,179.893,5.403,148.975
C04335=1217.334,-50.814,-39.486,179.896,5.404,148.975
C04336=1217.328,-50.565,-39.498,179.898,5.405,148.974
C04337=1217.324,-50.314,-39.511,179.900,5.404,148.973
C04338=1217.318,-50.065,-39.523,179.903,5.405,148.972
C04339=1217.313,-49.815,-39.535,179.905,5.405,148.972
C04340=1217.308,-49.565,-39.547,179.908,5.405,148.971
C04341=1217.303,-49.316,-39.560,179.910,5.405,148.970
C04342=1217.297,-49.046,-39.573,179.912,5.405,148.970
C04343=1217.292,-48.777,-39.586,179.916,5.405,148.969
C04344=1217.287,-48.506,-39.599,179.918,5.406,148.968
C04345=1217.281,-48.237,-39.611,179.921,5.406,148.967
C04346=1217.276,-47.987,-39.624,179.923,5.406,148.967
C04347=1217.271,-47.737,-39.637,179.926,5.406,148.966
C04348=1217.266,-47.487,-39.649,179.928,5.407,148.965
C04349=1217.260,-47.238,-39.662,179.930,5.406,148.964
C04350=1217.255,-46.988,-39.673,179.933,5.407,148.964
C04351=1217.250,-46.739,-39.686,179.935,5.407,148.963
C04352=1217.245,-46.489,-39.699,179.938,5.407,148.962
C04353=1217.240,-46.239,-39.711,179.940,5.408,148.962
C04354=1217.235,-45.989,-39.723,179.942,5.408,148.961
C04355=1217.230,-45.740,-39.736,179.945,5.408,148.960
C04356=1217.224,-45.490,-39.748,179.947,5.409,148.960
C04357=1217.219,-45.241,-39.761,179.950,5.408,148.959
C04358=1217.214,-44.991,-39.772,179.952,5.409,148.958
C04359=1217.209,-44.742,-39.785,179.954,5.408,148.958
C04360=1217.204,-44.492,-39.798,179.957,5.409,148.957
C04361=1217.199,-44.242,-39.811,179.960,5.409,148.956
C04362=1217.194,-43.992,-39.823,179.962,5.409,148.956
C04363=1217.188,-43.743,-39.835,179.964,5.409,148.955
C04364=1217.183,-43.494,-39.848,179.967,5.410,148.954
C04365=1217.178,-43.244,-39.860,179.969,5.410,148.953
C04366=1217.173,-42.994,-39.873,179.972,5.410,148.953
C04367=1217.168,-42.744,-39.885,179.974,5.411,148.952
C04368=1217.163,-42.495,-39.898,179.977,5.410,148.951
C04369=1217.157,-42.245,-39.910,179.979,5.411,148.951
C04370=1217.152,-41.996,-39.923,179.981,5.410,148.950
C04371=1217.147,-41.746,-39.936,179.984,5.411,148.949
C04372=1217.142,-41.496,-39.948,179.987,5.411,148.949
C04373=1217.137,-41.246,-39.960,179.988,5.411,148.948
C04374=1217.132,-40.997,-39.973,179.991,5.412,148.947
C04375=1217.127,-40.747,-39.986,179.994,5.412,148.947
C04376=1217.122,-40.498,-39.998,179.996,5.412,148.946
C04377=1217.117,-40.248,-40.011,179.998,5.412,148.945
C04378=1217.111,-39.998,-40.023,-179.999,5.413,148.945
C04379=1217.106,-39.749,-40.036,-179.997,5.413,148.944
C04380=1217.101,-39.499,-40.049,-179.994,5.413,148.943
C04381=1217.096,-39.249,-40.062,-179.992,5.414,148.942
C04382=1217.091,-39.000,-40.074,-179.990,5.413,148.942
C04383=1217.086,-38.751,-40.087,-179.987,5.414,148.941
C04384=1217.081,-38.500,-40.099,-179.984,5.414,148.940
C04385=1217.076,-38.251,-40.112,-179.982,5.414,148.940
C04386=1217.071,-38.002,-40.124,-179.979,5.414,148.939
C04387=1217.065,-37.752,-40.138,-179.977,5.414,148.938
C04388=1217.060,-37.502,-40.151,-179.975,5.414,148.938
C04389=1217.055,-37.253,-40.163,-179.972,5.415,148.937
C04390=1217.050,-37.003,-40.176,-179.970,5.415,148.936
C04391=1217.045,-36.754,-40.188,-179.967,5.415,148.935
C04392=1217.040,-36.503,-40.201,-179.965,5.416,148.935
C04393=1217.034,-36.254,-40.214,-179.963,5.415,148.934
C04394=1217.029,-36.004,-40.226,-179.960,5.416,148.934
C04395=1217.024,-35.754,-40.239,-179.958,5.417,148.933
C04396=1217.019,-35.505,-40.252,-179.956,5.416,148.932
C04397=1217.013,-35.255,-40.265,-179.953,5.417,148.931
C04398=1217.008,-35.006,-40.278,-179.950,5.417,148.931
C04399=1217.004,-34.756,-40.291,-179.948,5.417,148.930
C04400=1216.999,-34.507,-40.303,-179.946,5.417,148.929
C04401=1216.994,-34.257,-40.316,-179.943,5.418,148.929
C04402=1216.988,-34.007,-40.329,-179.941,5.418,148.928
C04403=1216.983,-33.758,-40.342,-179.938,5.418,148.927
C04404=1216.978,-33.508,-40.355,-179.936,5.418,148.927
C04405=1216.974,-33.258,-40.368,-179.933,5.418,148.926
C04406=1216.968,-33.009,-40.381,-179.931,5.419,148.925
C04407=1216.963,-32.759,-40.393,-179.928,5.419,148.924
C04408=1216.958,-32.509,-40.406,-179.926,5.419,148.924
C04409=1216.953,-32.260,-40.419,-179.923,5.419,148.923
C04410=1216.947,-32.011,-40.432,-179.921,5.420,148.922
C04411=1216.943,-31.760,-40.445,-179.919,5.419,148.922
C04412=1216.937,-31.511,-40.458,-179.916,5.420,148.921
C04413=1216.932,-31.262,-40.471,-179.913,5.420,148.920
C04414=1216.927,-31.012,-40.484,-179.911,5.420,148.920
C04415=1216.922,-30.763,-40.497,-179.909,5.421,148.919
C04416=1216.916,-30.513,-40.510,-179.906,5.421,148.918
C04417=1216.912,-30.263,-40.523,-179.904,5.421,148.918
C04418=1216.907,-30.014,-40.536,-179.902,5.422,148.917
C04419=1216.901,-29.764,-40.550,-179.899,5.422,148.916
C04420=1216.896,-29.514,-40.562,-179.896,5.423,148.916
C04421=1216.891,-29.265,-40.575,-179.894,5.422,148.915
C04422=1216.886,-29.015,-40.588,-179.892,5.423,148.914
C04423=1216.881,-28.766,-40.602,-179.889,5.423,148.914
C04424=1216.876,-28.517,-40.614,-179.887,5.423,148.913
C04425=1216.871,-28.266,-40.628,-179.884,5.423,148.912
C04426=1216.866,-28.017,-40.640,-179.882,5.424,148.911
C04427=1216.861,-27.767,-40.653,-179.879,5.424,148.911
C04428=1216.855,-27.517,-40.667,-179.877,5.424,148.910
C04429=1216.850,-27.269,-40.680,-179.874,5.425,148.909
C04430=1216.846,-27.019,-40.693,-179.872,5.424,148.909
C04431=1216.840,-26.769,-40.706,-179.869,5.425,148.908
C04432=1216.836,-26.519,-40.719,-179.867,5.425,148.907
C04433=1216.830,-26.269,-40.732,-179.865,5.425,148.907
C04434=1216.825,-26.020,-40.746,-179.862,5.425,148.906
C04435=1216.820,-25.771,-40.758,-179.859,5.426,148.905
C04436=1216.814,-25.521,-40.772,-179.857,5.427,148.905
C04437=1216.810,-25.271,-40.785,-179.855,5.426,148.904
C04438=1216.804,-25.022,-40.799,-179.852,5.427,148.903
C04439=1216.800,-24.772,-40.812,-179.850,5.427,148.903
C04440=1216.794,-24.522,-40.825,-179.848,5.427,148.902
C04441=1216.789,-24.272,-40.838,-179.845,5.428,148.901
C04442=1216.785,-24.024,-40.851,-179.842,5.428,148.901
C04443=1216.779,-23.773,-40.865,-179.840,5.428,148.900
C04444=1216.774,-23.524,-40.877,-179.838,5.428,148.899
C04445=1216.769,-23.274,-40.891,-179.835,5.429,148.898
C04446=1216.764,-23.005,-40.905,-179.832,5.429,148.898
C04447=1216.758,-22.736,-40.920,-179.830,5.429,148.897
C04448=1216.753,-22.466,-40.934,-179.827,5.429,148.896
C04449=1216.747,-22.197,-40.948,-179.824,5.429,148.895
C04450=1216.742,-21.947,-40.962,-179.822,5.430,148.895
C04451=1216.737,-21.698,-40.975,-179.819,5.430,148.894
C04452=1216.732,-21.448,-40.989,-179.817,5.430,148.893
C04453=1216.727,-21.199,-41.001,-179.814,5.431,148.893
C04454=1216.722,-20.949,-41.015,-179.812,5.431,148.892
C04455=1216.716,-20.699,-41.029,-179.810,5.431,148.892
C04456=1216.711,-20.449,-41.042,-179.807,5.432,148.891
C04457=1216.706,-20.200,-41.055,-179.805,5.432,148.890
C04458=1216.701,-19.950,-41.068,-179.802,5.433,148.889
C04459=1216.696,-19.701,-41.082,-179.800,5.432,148.889
C04460=1216.691,-19.451,-41.095,-179.797,5.433,148.888
C04461=1216.686,-19.202,-41.109,-179.795,5.433,148.887
C04462=1216.681,-18.952,-41.122,-179.793,5.433,148.887
C04463=1216.675,-18.703,-41.135,-179.790,5.434,148.886
C04464=1216.670,-18.453,-41.150,-179.787,5.434,148.885
C04465=1216.666,-18.203,-41.163,-179.785,5.435,148.885
C04466=1216.660,-17.954,-41.177,-179.783,5.434,148.884
C04467=1216.656,-17.704,-41.189,-179.780,5.435,148.883
C04468=1216.650,-17.455,-41.203,-179.777,5.435,148.882
C04469=1216.646,-17.205,-41.216,-179.775,5.435,148.882
C04470=1216.640,-16.956,-41.230,-179.773,5.435,148.881
C04471=1216.635,-16.705,-41.244,-179.770,5.436,148.880
C04472=1216.630,-16.457,-41.257,-179.767,5.436,148.880
C04473=1216.625,-16.206,-41.271,-179.765,5.436,148.879
C04474=1216.619,-15.957,-41.285,-179.763,5.437,148.879
C04475=1216.615,-15.707,-41.298,-179.760,5.437,148.878
C04476=1216.610,-15.458,-41.312,-179.758,5.438,148.877
C04477=1216.605,-15.209,-41.325,-179.756,5.438,148.876
C04478=1216.600,-14.959,-41.339,-179.753,5.438,148.876
C04479=1216.594,-14.710,-41.353,-179.750,5.439,148.875
C04480=1216.590,-14.460,-41.366,-179.748,5.439,148.874
C04481=1216.585,-14.210,-41.380,-179.746,5.439,148.874
C04482=1216.579,-13.960,-41.393,-179.743,5.439,148.873
C04483=1216.575,-13.711,-41.407,-179.740,5.440,148.872
C04484=1216.569,-13.462,-41.421,-179.738,5.439,148.872
C04485=1216.564,-13.212,-41.434,-179.735,5.440,148.871
C04486=1216.560,-12.962,-41.448,-179.733,5.440,148.870
C04487=1216.554,-12.713,-41.462,-179.730,5.441,148.870
C04488=1216.549,-12.463,-41.475,-179.728,5.441,148.869
C04489=1216.543,-12.214,-41.489,-179.725,5.441,148.868
C04490=1216.539,-11.964,-41.503,-179.723,5.442,148.867
C04491=1216.534,-11.714,-41.517,-179.720,5.442,148.867
C04492=1216.528,-11.465,-41.530,-179.719,5.442,148.866
C04493=1216.524,-11.216,-41.544,-179.716,5.443,148.866
C04494=1216.519,-10.965,-41.558,-179.713,5.443,148.865
C04495=1216.513,-10.716,-41.572,-179.711,5.444,148.864
C04496=1216.508,-10.467,-41.586,-179.709,5.443,148.864
C04497=1216.504,-10.217,-41.599,-179.706,5.444,148.863
C04498=1216.498,-9.968,-41.613,-179.703,5.444,148.862
C04499=1216.493,-9.718,-41.627,-179.701,5.445,148.861
C04500=1216.488,-9.468,-41.641,-179.698,5.445,148.861
C04501=1216.483,-9.219,-41.654,-179.696,5.445,148.860
C04502=1216.478,-8.969,-41.668,-179.693,5.446,148.859
C04503=1216.473,-8.719,-41.683,-179.690,5.446,148.859
C04504=1216.468,-8.470,-41.696,-179.688,5.446,148.858
C04505=1216.462,-8.220,-41.710,-179.686,5.446,148.857
C04506=1216.458,-7.971,-41.724,-179.683,5.447,148.857
C04507=1216.453,-7.722,-41.738,-179.680,5.447,148.856
C04508=1216.448,-7.472,-41.752,-179.678,5.447,148.855
C04509=1216.443,-7.222,-41.766,-179.676,5.448,148.855
C04510=1216.437,-6.973,-41.779,-179.674,5.448,148.854
C04511=1216.433,-6.723,-41.793,-179.671,5.449,148.853
C04512=1216.428,-6.473,-41.807,-179.669,5.449,148.853
C04513=1216.423,-6.224,-41.822,-179.666,5.449,148.852
C04514=1216.417,-5.975,-41.835,-179.664,5.450,148.851
C04515=1216.412,-5.725,-41.850,-179.661,5.450,148.851
C04516=1216.407,-5.475,-41.863,-179.658,5.451,148.850
C04517=1216.402,-5.226,-41.877,-179.656,5.450,148.849
C04518=1216.397,-4.976,-41.891,-179.653,5.451,148.849
C04519=1216.392,-4.727,-41.905,-179.651,5.451,148.848
C04520=1216.387,-4.477,-41.919,-179.648,5.452,148.847
C04521=1216.382,-4.228,-41.933,-179.646,5.452,148.846
C04522=1216.377,-3.978,-41.948,-179.643,5.452,148.846
C04523=1216.372,-3.728,-41.962,-179.641,5.453,148.845
C04524=1216.367,-3.479,-41.976,-179.639,5.453,148.845
C04525=1216.361,-3.229,-41.989,-179.636,5.454,148.844
C04526=1216.357,-2.980,-42.003,-179.634,5.454,148.843
C04527=1216.352,-2.730,-42.017,-179.631,5.454,148.843
C04528=1216.347,-2.480,-42.032,-179.629,5.455,148.842
C04529=1216.341,-2.231,-42.046,-179.626,5.455,148.841
C04530=1216.336,-1.982,-42.060,-179.624,5.455,148.840
C04531=1216.331,-1.732,-42.074,-179.621,5.455,148.840
C04532=1216.326,-1.482,-42.088,-179.619,5.456,148.839
C04533=1216.321,-1.232,-42.103,-179.616,5.456,148.838
C04534=1216.316,-0.983,-42.117,-179.613,5.457,148.838
C04535=1216.311,-0.734,-42.131,-179.611,5.457,148.837
C04536=1216.306,-0.484,-42.145,-179.608,5.457,148.836
C04537=1216.301,-0.234,-42.159,-179.606,5.458,148.836
C04538=1216.296,0.015,-42.174,-179.603,5.458,148.835
C04539=1216.290,0.264,-42.188,-179.602,5.458,148.835
C04540=1216.286,0.514,-42.202,-179.599,5.459,148.834
C04541=1216.281,0.764,-42.216,-179.596,5.459,148.833
C04542=1216.276,1.014,-42.230,-179.594,5.460,148.832
C04543=1216.271,1.263,-42.245,-179.591,5.460,148.832
C04544=1216.265,1.512,-42.259,-179.589,5.460,148.831
C04545=1216.260,1.761,-42.274,-179.586,5.460,148.830
C04546=1216.255,2.011,-42.288,-179.584,5.461,148.830
C04547=1216.251,2.261,-42.302,-179.581,5.461,148.829
C04548=1216.246,2.510,-42.316,-179.578,5.462,148.828
C04549=1216.241,2.760,-42.331,-179.576,5.462,148.828
C04550=1216.235,3.028,-42.346,-179.574,5.462,148.827
C04551=1216.229,3.298,-42.361,-179.571,5.463,148.826
C04552=1216.224,3.566,-42.377,-179.568,5.463,148.826
C04553=1216.218,3.836,-42.393,-179.566,5.464,148.825
C04554=1216.214,4.085,-42.407,-179.563,5.464,148.824
C04555=1216.209,4.335,-42.422,-179.560,5.465,148.824
C04556=1216.204,4.585,-42.436,-179.558,5.465,148.823
C04557=1216.199,4.834,-42.450,-179.556,5.465,148.822
C04558=1216.193,5.083,-42.464,-179.553,5.466,148.821
C04559=1216.188,5.333,-42.479,-179.550,5.466,148.821
C04560=1216.183,5.582,-42.493,-179.548,5.467,148.820
C04561=1216.179,5.832,-42.508,-179.545,5.467,148.819
C04562=1216.174,6.082,-42.522,-179.542,5.468,148.819
C04563=1216.169,6.331,-42.537,-179.540,5.467,148.818
C04564=1216.163,6.581,-42.552,-179.538,5.468,148.818
C04565=1216.158,6.830,-42.566,-179.535,5.469,148.817
C04566=1216.153,7.080,-42.580,-179.533,5.469,148.816
C04567=1216.148,7.329,-42.595,-179.530,5.470,148.815
C04568=1216.143,7.578,-42.609,-179.528,5.469,148.815
C04569=1216.138,7.828,-42.623,-179.525,5.470,148.814
C04570=1216.133,8.078,-42.638,-179.523,5.470,148.813
C04571=1216.128,8.327,-42.653,-179.520,5.471,148.813
C04572=1216.123,8.577,-42.668,-179.517,5.471,148.812
C04573=1216.118,8.827,-42.682,-179.515,5.472,148.811
C04574=1216.113,9.076,-42.697,-179.513,5.472,148.811
C04575=1216.108,9.325,-42.711,-179.510,5.472,148.810
C04576=1216.103,9.575,-42.725,-179.508,5.473,148.810
C04577=1216.098,9.824,-42.741,-179.505,5.474,148.809
C04578=1216.093,10.074,-42.755,-179.503,5.474,148.808
C04579=1216.088,10.324,-42.770,-179.500,5.475,148.807
C04580=1216.083,10.573,-42.785,-179.498,5.474,148.807
C04581=1216.078,10.823,-42.799,-179.495,5.475,148.806
C04582=1216.073,11.073,-42.814,-179.493,5.475,148.805
C04583=1216.068,11.322,-42.829,-179.490,5.476,148.805
C04584=1216.063,11.571,-42.843,-179.487,5.476,148.804
C04585=1216.058,11.820,-42.858,-179.485,5.477,148.803
C04586=1216.052,12.070,-42.873,-179.483,5.477,148.803
C04587=1216.047,12.320,-42.887,-179.480,5.478,148.802
C04588=1216.043,12.569,-42.902,-179.478,5.478,148.802
C04589=1216.038,12.818,-42.916,-179.475,5.479,148.801
C04590=1216.032,13.068,-42.932,-179.472,5.479,148.800
C04591=1216.027,13.318,-42.946,-179.470,5.480,148.800
C04592=1216.023,13.567,-42.961,-179.468,5.479,148.799
C04593=1216.017,13.817,-42.976,-179.465,5.480,148.798
C04594=1216.012,14.066,-42.991,-179.462,5.480,148.797
C04595=1216.007,14.315,-43.005,-179.460,5.481,148.797
C04596=1216.003,14.565,-43.020,-179.457,5.481,148.796
C04597=1215.997,14.815,-43.035,-179.455,5.482,148.796
C04598=1215.992,15.064,-43.050,-179.452,5.483,148.795
C04599=1215.987,15.313,-43.064,-179.450,5.483,148.794
C04600=1215.983,15.563,-43.080,-179.448,5.483,148.794
C04601=1215.978,15.813,-43.094,-179.445,5.484,148.793
C04602=1215.973,16.062,-43.109,-179.442,5.484,148.792
C04603=1215.967,16.312,-43.124,-179.440,5.485,148.792
C04604=1215.963,16.561,-43.139,-179.437,5.485,148.791
C04605=1215.958,16.811,-43.154,-179.434,5.486,148.790
C04606=1215.952,17.061,-43.169,-179.432,5.485,148.789
C04607=1215.948,17.310,-43.184,-179.430,5.486,148.789
C04608=1215.942,17.560,-43.199,-179.428,5.487,148.788
C04609=1215.937,17.809,-43.214,-179.425,5.487,148.788
C04610=1215.932,18.058,-43.228,-179.422,5.488,148.787
C04611=1215.927,18.308,-43.244,-179.420,5.488,148.786
C04612=1215.922,18.557,-43.259,-179.417,5.489,148.786
C04613=1215.917,18.807,-43.274,-179.415,5.489,148.785
C04614=1215.912,19.056,-43.289,-179.412,5.489,148.784
C04615=1215.907,19.305,-43.304,-179.410,5.490,148.784
C04616=1215.902,19.556,-43.319,-179.407,5.490,148.783
C04617=1215.898,19.805,-43.334,-179.405,5.491,148.782
C04618=1215.892,20.055,-43.349,-179.402,5.492,148.782
C04619=1215.887,20.304,-43.364,-179.399,5.492,148.781
C04620=1215.883,20.553,-43.379,-179.397,5.493,148.780
C04621=1215.877,20.803,-43.394,-179.395,5.492,148.780
C04622=1215.872,21.052,-43.409,-179.392,5.493,148.779
C04623=1215.867,21.302,-43.424,-179.389,5.494,148.778
C04624=1215.862,21.551,-43.439,-179.387,5.494,148.778
C04625=1215.857,21.801,-43.454,-179.384,5.495,148.777
C04626=1215.853,22.051,-43.469,-179.382,5.495,148.777
C04627=1215.847,22.300,-43.485,-179.379,5.496,148.776
C04628=1215.843,22.549,-43.500,-179.377,5.497,148.775
C04629=1215.837,22.799,-43.515,-179.375,5.496,148.774
C04630=1215.832,23.048,-43.530,-179.372,5.497,148.774
C04631=1215.827,23.298,-43.546,-179.369,5.497,148.773
C04632=1215.822,23.547,-43.561,-179.367,5.498,148.772
C04633=1215.817,23.797,-43.576,-179.364,5.498,148.772
C04634=1215.812,24.046,-43.591,-179.361,5.499,148.771
C04635=1215.807,24.296,-43.606,-179.359,5.500,148.771
C04636=1215.802,24.545,-43.621,-179.357,5.500,148.770
C04637=1215.797,24.794,-43.637,-179.354,5.501,148.769
C04638=1215.792,25.043,-43.652,-179.352,5.501,148.769
C04639=1215.787,25.294,-43.667,-179.349,5.501,148.768
C04640=1215.783,25.543,-43.682,-179.347,5.502,148.767
C04641=1215.777,25.793,-43.698,-179.344,5.502,148.767
C04642=1215.772,26.042,-43.713,-179.341,5.503,148.766
C04643=1215.767,26.291,-43.728,-179.339,5.504,148.765
C04644=1215.762,26.541,-43.744,-179.337,5.504,148.765
C04645=1215.758,26.790,-43.759,-179.334,5.505,148.764
C04646=1215.752,27.040,-43.775,-179.331,5.505,148.763
C04647=1215.748,27.289,-43.790,-179.329,5.506,148.763
C04648=1215.742,27.539,-43.805,-179.326,5.506,148.762
C04649=1215.737,27.789,-43.821,-179.324,5.506,148.761
C04650=1215.733,28.038,-43.836,-179.321,5.507,148.761
C04651=1215.727,28.287,-43.851,-179.319,5.507,148.760
C04652=1215.722,28.537,-43.867,-179.316,5.508,148.760
C04653=1215.717,28.786,-43.882,-179.314,5.508,148.759
C04654=1215.712,29.055,-43.899,-179.311,5.509,148.758
C04655=1215.706,29.324,-43.916,-179.308,5.510,148.758
C04656=1215.701,29.592,-43.932,-179.306,5.510,148.757
C04657=1215.696,29.861,-43.949,-179.303,5.510,148.756
C04658=1215.691,30.110,-43.965,-179.301,5.511,148.755
C04659=1215.686,30.359,-43.980,-179.298,5.512,148.755
C04660=1215.681,30.609,-43.995,-179.295,5.512,148.754
C04661=1215.676,30.859,-44.011,-179.293,5.513,148.753
C04662=1215.671,31.108,-44.026,-179.290,5.513,148.753
C04663=1215.666,31.357,-44.042,-179.287,5.514,148.752
C04664=1215.661,31.607,-44.058,-179.285,5.514,148.751
C04665=1215.656,31.857,-44.073,-179.283,5.515,148.751
C04666=1215.651,32.106,-44.088,-179.280,5.516,148.750
C04667=1215.646,32.356,-44.104,-179.277,5.516,148.750
C04668=1215.641,32.605,-44.120,-179.275,5.516,148.749
C04669=1215.636,32.855,-44.135,-179.273,5.517,148.748
C04670=1215.631,33.104,-44.150,-179.270,5.517,148.748
C04671=1215.626,33.353,-44.167,-179.267,5.518,148.747
C04672=1215.622,33.603,-44.182,-179.265,5.519,148.746
C04673=1215.616,33.852,-44.198,-179.262,5.519,148.746
C04674=1215.611,34.102,-44.214,-179.260,5.520,148.745
C04675=1215.606,34.351,-44.229,-179.257,5.520,148.744
C04676=1215.601,34.601,-44.244,-179.255,5.521,148.744
C04677=1215.597,34.851,-44.260,-179.252,5.521,148.743
C04678=1215.591,35.099,-44.276,-179.249,5.522,148.742
C04679=1215.586,35.349,-44.292,-179.247,5.523,148.742
C04680=1215.581,35.599,-44.308,-179.244,5.523,148.741
C04681=1215.577,35.848,-44.323,-179.242,5.524,148.741
C04682=1215.571,36.097,-44.338,-179.239,5.524,148.740
C04683=1215.566,36.348,-44.354,-179.237,5.525,148.739
C04684=1215.561,36.596,-44.371,-179.234,5.525,148.739
C04685=1215.556,36.846,-44.386,-179.232,5.525,148.738
C04686=1215.552,37.096,-44.402,-179.230,5.526,148.737
C04687=1215.547,37.345,-44.417,-179.227,5.527,148.737
C04688=1215.541,37.594,-44.434,-179.224,5.527,148.736
C04689=1215.537,37.844,-44.450,-179.222,5.528,148.735
C04690=1215.531,38.093,-44.465,-179.219,5.528,148.735
C04691=1215.526,38.343,-44.481,-179.216,5.529,148.734
C04692=1215.521,38.592,-44.497,-179.214,5.530,148.734
C04693=1215.517,38.841,-44.512,-179.212,5.530,148.733
C04694=1215.512,39.091,-44.528,-179.209,5.531,148.732
C04695=1215.507,39.340,-44.545,-179.206,5.531,148.732
C04696=1215.502,39.589,-44.560,-179.204,5.532,148.731
C04697=1215.497,39.840,-44.576,-179.201,5.532,148.730
C04698=1215.492,40.088,-44.592,-179.198,5.533,148.730
C04699=1215.487,40.338,-44.608,-179.196,5.534,148.729
C04700=1215.481,40.588,-44.624,-179.194,5.534,148.728
C04701=1215.476,40.837,-44.640,-179.191,5.535,148.728
C04702=1215.472,41.086,-44.656,-179.188,5.535,148.727
C04703=1215.467,41.336,-44.671,-179.186,5.536,148.726
C04704=1215.462,41.585,-44.688,-179.183,5.537,148.726
C04705=1215.457,41.835,-44.704,-179.181,5.537,148.725
C04706=1215.452,42.084,-44.720,-179.178,5.538,148.725
C04707=1215.447,42.334,-44.736,-179.176,5.539,148.724
C04708=1215.442,42.583,-44.751,-179.173,5.539,148.723
C04709=1215.437,42.833,-44.768,-179.170,5.540,148.723
C04710=1215.432,43.082,-44.784,-179.168,5.540,148.722
C04711=1215.428,43.331,-44.800,-179.166,5.541,148.722
C04712=1215.422,43.581,-44.816,-179.163,5.542,148.721
C04713=1215.418,43.830,-44.833,-179.161,5.541,148.720
C04714=1215.412,44.080,-44.848,-179.158,5.542,148.720
C04715=1215.407,44.330,-44.864,-179.156,5.543,148.719
C04716=1215.402,44.579,-44.880,-179.153,5.543,148.718
C04717=1215.397,44.828,-44.896,-179.151,5.544,148.718
C04718=1215.393,45.077,-44.913,-179.148,5.545,148.717
C04719=1215.387,45.327,-44.928,-179.146,5.545,148.716
C04720=1215.383,45.576,-44.945,-179.143,5.546,148.716
C04721=1215.378,45.825,-44.961,-179.140,5.546,148.715
C04722=1215.373,46.075,-44.977,-179.138,5.547,148.715
C04723=1215.368,46.324,-44.993,-179.136,5.548,148.714
C04724=1215.363,46.574,-45.009,-179.133,5.548,148.713
C04725=1215.358,46.823,-45.026,-179.130,5.549,148.713
C04726=1215.353,47.073,-45.042,-179.128,5.549,148.712
C04727=1215.348,47.322,-45.058,-179.125,5.550,148.711
C04728=1215.343,47.572,-45.074,-179.123,5.551,148.711
C04729=1215.338,47.821,-45.090,-179.120,5.551,148.710
C04730=1215.333,48.070,-45.107,-179.118,5.552,148.709
C04731=1215.328,48.321,-45.123,-179.115,5.552,148.709
C04732=1215.323,48.569,-45.140,-179.112,5.553,148.708
C04733=1215.318,48.819,-45.156,-179.110,5.554,148.708
C04734=1215.313,49.068,-45.172,-179.107,5.554,148.707
C04735=1215.309,49.318,-45.189,-179.105,5.555,148.706
C04736=1215.303,49.567,-45.204,-179.102,5.556,148.706
C04737=1215.299,49.817,-45.221,-179.100,5.556,148.705
C04738=1215.294,50.065,-45.237,-179.097,5.557,148.705
C04739=1215.289,50.316,-45.253,-179.095,5.558,148.704
C04740=1215.283,50.565,-45.270,-179.092,5.558,148.703
C04741=1215.279,50.814,-45.287,-179.090,5.559,148.703
C04742=1215.274,51.064,-45.303,-179.087,5.559,148.702
C04743=1215.269,51.313,-45.319,-179.084,5.561,148.701
C04744=1215.264,51.562,-45.336,-179.082,5.561,148.701
C04745=1215.259,51.811,-45.352,-179.079,5.562,148.700
C04746=1215.254,52.062,-45.369,-179.076,5.563,148.699
C04747=1215.249,52.311,-45.385,-179.074,5.563,148.699
C04748=1215.244,52.560,-45.402,-179.071,5.564,148.698
C04749=1215.240,52.809,-45.418,-179.069,5.565,148.698
C04750=1215.234,53.059,-45.434,-179.066,5.565,148.697
C04751=1215.230,53.308,-45.450,-179.064,5.566,148.696
C04752=1215.225,53.558,-45.468,-179.061,5.566,148.696
C04753=1215.219,53.807,-45.484,-179.059,5.567,148.695
C04754=1215.215,54.056,-45.501,-179.056,5.568,148.695
C04755=1215.210,54.306,-45.516,-179.054,5.568,148.694
C04756=1215.204,54.556,-45.534,-179.051,5.569,148.693
C04757=1215.200,54.805,-45.550,-179.048,5.569,148.693
C04758=1215.195,55.073,-45.568,-179.046,5.570,148.692
C04759=1215.189,55.341,-45.585,-179.043,5.571,148.691
C04760=1215.184,55.610,-45.604,-179.040,5.571,148.691
C04761=1215.178,55.878,-45.621,-179.037,5.572,148.690
C04762=1215.174,56.128,-45.638,-179.035,5.573,148.689
C04763=1215.169,56.377,-45.655,-179.032,5.574,148.689
C04764=1215.163,56.627,-45.671,-179.030,5.574,148.688
C04765=1215.159,56.876,-45.688,-179.027,5.575,148.687
C04766=1215.154,57.126,-45.705,-179.024,5.576,148.687
C04767=1215.149,57.375,-45.721,-179.022,5.577,148.686
C04768=1215.144,57.624,-45.738,-179.020,5.577,148.686
C04769=1215.139,57.874,-45.755,-179.017,5.578,148.685
C04770=1215.134,58.123,-45.771,-179.014,5.578,148.684
C04771=1215.129,58.372,-45.788,-179.012,5.579,148.684
C04772=1215.124,58.622,-45.805,-179.010,5.580,148.683
C04773=1215.119,58.871,-45.822,-179.007,5.580,148.683
C04774=1215.115,59.120,-45.838,-179.004,5.581,148.682
C04775=1215.109,59.370,-45.856,-179.002,5.581,148.681
C04776=1215.104,59.619,-45.872,-179.000,5.582,148.681
C04777=1215.100,59.869,-45.889,-178.996,5.584,148.680
C04778=1215.095,60.118,-45.906,-178.994,5.584,148.679
C04779=1215.090,60.368,-45.922,-178.991,5.585,148.679
C04780=1215.085,60.617,-45.939,-178.989,5.586,148.678
C04781=1215.080,60.866,-45.956,-178.986,5.586,148.678
C04782=1215.075,61.116,-45.973,-178.984,5.587,148.677
C04783=1215.069,61.365,-45.990,-178.981,5.587,148.676
C04784=1215.065,61.614,-46.006,-178.979,5.588,148.676
C04785=1215.061,61.864,-46.023,-178.976,5.589,148.675
C04786=1215.055,62.114,-46.040,-178.974,5.589,148.675
C04787=1215.050,62.362,-46.056,-178.971,5.590,148.674
C04788=1215.045,62.612,-46.074,-178.968,5.591,148.673
C04789=1215.041,62.861,-46.091,-178.966,5.591,148.673
C04790=1215.036,63.111,-46.108,-178.964,5.592,148.672
C04791=1215.031,63.360,-46.125,-178.961,5.593,148.672
C04792=1215.026,63.609,-46.141,-178.958,5.594,148.671
C04793=1215.021,63.859,-46.159,-178.956,5.595,148.670
C04794=1215.016,64.109,-46.175,-178.953,5.595,148.670
C04795=1215.011,64.358,-46.193,-178.950,5.596,148.669
C04796=1215.006,64.606,-46.210,-178.948,5.597,148.668
C04797=1215.001,64.856,-46.227,-178.946,5.598,148.668
C04798=1214.997,65.106,-46.244,-178.943,5.598,148.667
C04799=1214.991,65.356,-46.261,-178.940,5.599,148.667
C04800=1214.987,65.605,-46.277,-178.938,5.599,148.666
C04801=1214.981,65.853,-46.295,-178.936,5.600,148.666
C04802=1214.977,66.103,-46.312,-178.933,5.601,148.665
C04803=1214.972,66.353,-46.329,-178.930,5.602,148.664
C04804=1214.967,66.602,-46.346,-178.927,5.603,148.664
C04805=1214.962,66.851,-46.364,-178.925,5.604,148.663
C04806=1214.957,67.100,-46.380,-178.922,5.604,148.663
C04807=1214.952,67.350,-46.397,-178.920,5.605,148.662
C04808=1214.948,67.599,-46.414,-178.917,5.605,148.661
C04809=1214.943,67.849,-46.432,-178.915,5.606,148.661
C04810=1214.937,68.098,-46.449,-178.912,5.607,148.660
C04811=1214.933,68.348,-46.466,-178.910,5.607,148.659
C04812=1214.927,68.596,-46.483,-178.907,5.608,148.659
C04813=1214.923,68.846,-46.500,-178.904,5.610,148.658
C04814=1214.918,69.096,-46.517,-178.902,5.610,148.658
C04815=1214.914,69.345,-46.535,-178.899,5.611,148.657
C04816=1214.908,69.594,-46.552,-178.896,5.611,148.656
C04817=1214.903,69.844,-46.569,-178.894,5.612,148.656
C04818=1214.899,70.093,-46.587,-178.892,5.613,148.655
C04819=1214.893,70.342,-46.604,-178.889,5.613,148.655
C04820=1214.889,70.592,-46.620,-178.887,5.614,148.654
C04821=1214.884,70.841,-46.638,-178.884,5.615,148.654
C04822=1214.879,71.091,-46.655,-178.881,5.616,148.653
C04823=1214.874,71.339,-46.673,-178.878,5.617,148.652
C04824=1214.869,71.589,-46.690,-178.876,5.618,148.652
C04825=1214.864,71.839,-46.707,-178.874,5.618,148.651
C04826=1214.860,72.088,-46.725,-178.871,5.619,148.650
C04827=1214.855,72.338,-46.742,-178.868,5.620,148.650
C04828=1214.849,72.586,-46.760,-178.866,5.620,148.649
C04829=1214.845,72.836,-46.776,-178.864,5.621,148.649
C04830=1214.840,73.085,-46.794,-178.860,5.622,148.648
C04831=1214.834,73.335,-46.812,-178.858,5.623,148.648
C04832=1214.830,73.583,-46.829,-178.856,5.624,148.647
C04833=1214.825,73.833,-46.846,-178.853,5.624,148.646
C04834=1214.820,74.082,-46.864,-178.850,5.625,148.646
C04835=1214.815,74.332,-46.881,-178.848,5.626,148.645
C04836=1214.811,74.581,-46.899,-178.846,5.627,148.645
C04837=1214.806,74.831,-46.916,-178.842,5.628,148.644
C04838=1214.801,75.080,-46.934,-178.840,5.629,148.643
C04839=1214.795,75.330,-46.951,-178.838,5.629,148.643
C04840=1214.791,75.579,-46.969,-178.835,5.630,148.642
C04841=1214.786,75.829,-46.986,-178.832,5.631,148.641
C04842=1214.781,76.078,-47.004,-178.830,5.632,148.641
C04843=1214.776,76.327,-47.022,-178.828,5.632,148.640
C04844=1214.772,76.576,-47.039,-178.824,5.634,148.640
C04845=1214.767,76.826,-47.057,-178.822,5.634,148.639
C04846=1214.761,77.075,-47.073,-178.820,5.635,148.639
C04847=1214.756,77.324,-47.091,-178.817,5.636,148.638
C04848=1214.752,77.573,-47.109,-178.815,5.637,148.638
C04849=1214.747,77.822,-47.126,-178.812,5.637,148.637
C04850=1214.742,78.072,-47.144,-178.810,5.638,148.636
C04851=1214.737,78.321,-47.162,-178.806,5.639,148.636
C04852=1214.732,78.571,-47.179,-178.804,5.640,148.635
C04853=1214.727,78.820,-47.197,-178.802,5.641,148.635
C04854=1214.723,79.069,-47.215,-178.799,5.641,148.634
C04855=1214.717,79.318,-47.232,-178.797,5.642,148.633
C04856=1214.712,79.568,-47.250,-178.794,5.643,148.633
C04857=1214.707,79.817,-47.268,-178.791,5.644,148.632
C04858=1214.703,80.067,-47.286,-178.789,5.645,148.632
C04859=1214.698,80.316,-47.304,-178.786,5.646,148.631
C04860=1214.694,80.565,-47.321,-178.784,5.646,148.630
C04861=1214.689,80.815,-47.339,-178.781,5.647,148.630
C04862=1214.683,81.083,-47.358,-178.778,5.648,148.629
C04863=1214.678,81.351,-47.377,-178.776,5.649,148.629
C04864=1214.673,81.619,-47.396,-178.773,5.650,148.628
C04865=1214.667,81.888,-47.415,-178.770,5.651,148.627
C04866=1214.662,82.137,-47.433,-178.767,5.652,148.627
C04867=1214.658,82.386,-47.451,-178.765,5.653,148.626
C04868=1214.653,82.636,-47.469,-178.763,5.653,148.626
C04869=1214.647,82.885,-47.486,-178.760,5.654,148.625
C04870=1214.643,83.135,-47.504,-178.757,5.655,148.625
C04871=1214.638,83.384,-47.522,-178.755,5.656,148.624
C04872=1214.633,83.634,-47.540,-178.752,5.657,148.623
C04873=1214.628,83.883,-47.558,-178.749,5.657,148.623
C04874=1214.623,84.132,-47.576,-178.747,5.658,148.622
C04875=1214.619,84.381,-47.594,-178.745,5.659,148.622
C04876=1214.613,84.631,-47.611,-178.741,5.660,148.621
C04877=1214.608,84.880,-47.629,-178.739,5.661,148.620
C04878=1214.603,85.129,-47.647,-178.737,5.662,148.620
C04879=1214.599,85.378,-47.665,-178.734,5.662,148.619
C04880=1214.594,85.628,-47.683,-178.732,5.663,148.619
C04881=1214.589,85.878,-47.702,-178.729,5.665,148.618
C04882=1214.584,86.127,-47.720,-178.726,5.665,148.617
C04883=1214.580,86.376,-47.738,-178.724,5.666,148.617
C04884=1214.575,86.625,-47.756,-178.721,5.667,148.616
C04885=1214.570,86.874,-47.774,-178.719,5.667,148.616
C04886=1214.565,87.123,-47.792,-178.716,5.669,148.615
C04887=1214.560,87.373,-47.810,-178.713,5.670,148.615
C04888=1214.556,87.622,-47.828,-178.711,5.671,148.614
C04889=1214.551,87.872,-47.846,-178.709,5.671,148.614
C04890=1214.546,88.121,-47.864,-178.706,5.672,148.613
C04891=1214.541,88.370,-47.882,-178.703,5.673,148.612
C04892=1214.536,88.619,-47.900,-178.701,5.674,148.612
C04893=1214.531,88.868,-47.918,-178.698,5.675,148.611
C04894=1214.527,89.118,-47.936,-178.696,5.676,148.611
C04895=1214.522,89.367,-47.954,-178.693,5.677,148.610
C04896=1214.517,89.617,-47.972,-178.690,5.678,148.609
C04897=1214.512,89.866,-47.990,-178.688,5.678,148.609
C04898=1214.506,90.115,-48.009,-178.685,5.679,148.608
C04899=1214.501,90.364,-48.027,-178.683,5.680,148.608
C04900=1214.497,90.614,-48.045,-178.680,5.681,148.607
C04901=1214.492,90.863,-48.063,-178.677,5.682,148.607
C04902=1214.487,91.113,-48.081,-178.675,5.683,148.606
C04903=1214.483,91.361,-48.100,-178.673,5.684,148.606
C04904=1214.478,91.610,-48.118,-178.670,5.685,148.605
C04905=1214.473,91.861,-48.137,-178.667,5.686,148.605
C04906=1214.468,92.110,-48.155,-178.665,5.686,148.604
C04907=1214.463,92.359,-48.173,-178.662,5.687,148.603
C04908=1214.458,92.608,-48.191,-178.660,5.688,148.603
C04909=1214.454,92.857,-48.210,-178.657,5.689,148.602
C04910=1214.449,93.107,-48.228,-178.654,5.690,148.602
C04911=1214.443,93.356,-48.246,-178.652,5.691,148.601
C04912=1214.438,93.605,-48.264,-178.649,5.692,148.600
C04913=1214.434,93.855,-48.282,-178.646,5.693,148.600
C04914=1214.430,94.104,-48.301,-178.644,5.694,148.599
C04915=1214.425,94.353,-48.319,-178.641,5.694,148.599
C04916=1214.419,94.602,-48.338,-178.639,5.695,148.598
C04917=1214.415,94.852,-48.356,-178.636,5.697,148.598
C04918=1214.410,95.101,-48.375,-178.634,5.697,148.597
C04919=1214.405,95.350,-48.393,-178.631,5.698,148.597
C04920=1214.400,95.599,-48.411,-178.629,5.699,148.596
C04921=1214.395,95.849,-48.430,-178.626,5.700,148.595
C04922=1214.391,96.098,-48.448,-178.623,5.701,148.595
C04923=1214.386,96.347,-48.466,-178.621,5.702,148.594
C04924=1214.381,96.597,-48.485,-178.619,5.703,148.594
C04925=1214.376,96.846,-48.504,-178.616,5.704,148.593
C04926=1214.371,97.095,-48.522,-178.613,5.705,148.593
C04927=1214.366,97.344,-48.540,-178.611,5.706,148.592
C04928=1214.361,97.594,-48.560,-178.608,5.707,148.591
C04929=1214.357,97.843,-48.578,-178.605,5.708,148.591
C04930=1214.352,98.092,-48.596,-178.603,5.709,148.590
C04931=1214.347,98.342,-48.615,-178.600,5.709,148.590
C04932=1214.342,98.591,-48.633,-178.598,5.711,148.589
C04933=1214.337,98.839,-48.652,-178.595,5.712,148.589
C04934=1214.332,99.089,-48.671,-178.593,5.713,148.588
C04935=1214.327,99.339,-48.689,-178.590,5.713,148.588
C04936=1214.323,99.587,-48.708,-178.587,5.715,148.587
C04937=1214.318,99.837,-48.726,-178.585,5.716,148.587
C04938=1214.313,100.086,-48.745,-178.582,5.716,148.586
C04939=1214.308,100.335,-48.763,-178.580,5.717,148.586
C04940=1214.303,100.585,-48.783,-178.577,5.719,148.585
C04941=1214.299,100.834,-48.801,-178.574,5.719,148.584
C04942=1214.293,101.083,-48.820,-178.572,5.720,148.584
C04943=1214.289,101.333,-48.838,-178.569,5.721,148.583
C04944=1214.284,101.581,-48.857,-178.567,5.722,148.583
C04945=1214.279,101.831,-48.876,-178.564,5.723,148.582
C04946=1214.275,102.080,-48.895,-178.562,5.724,148.581
C04947=1214.269,102.329,-48.913,-178.559,5.725,148.581
C04948=1214.265,102.579,-48.932,-178.556,5.726,148.580
C04949=1214.260,102.828,-48.950,-178.554,5.727,148.580
C04950=1214.255,103.077,-48.970,-178.551,5.728,148.579
C04951=1214.250,103.327,-48.988,-178.548,5.729,148.579
C04952=1214.245,103.575,-49.007,-178.546,5.730,148.578
C04953=1214.241,103.825,-49.026,-178.543,5.731,148.578
C04954=1214.235,104.074,-49.045,-178.541,5.732,148.577
C04955=1214.231,104.323,-49.064,-178.538,5.733,148.577
C04956=1214.226,104.573,-49.083,-178.536,5.734,148.576
C04957=1214.221,104.821,-49.101,-178.533,5.735,148.576
C04958=1214.216,105.071,-49.121,-178.530,5.736,148.575
C04959=1214.212,105.320,-49.139,-178.528,5.737,148.575
C04960=1214.207,105.570,-49.159,-178.525,5.738,148.574
C04961=1214.202,105.819,-49.177,-178.523,5.739,148.573
C04962=1214.197,106.069,-49.196,-178.520,5.740,148.573
C04963=1214.193,106.317,-49.215,-178.518,5.742,148.572
C04964=1214.188,106.567,-49.235,-178.515,5.742,148.572
C04965=1214.183,106.816,-49.253,-178.512,5.743,148.571
C04966=1214.177,107.084,-49.273,-178.510,5.744,148.571
C04967=1214.172,107.353,-49.294,-178.507,5.745,148.570
C04968=1214.167,107.621,-49.314,-178.504,5.746,148.569
C04969=1214.162,107.889,-49.335,-178.501,5.747,148.569
C04970=1214.157,108.139,-49.353,-178.499,5.749,148.568
C04971=1214.153,108.388,-49.372,-178.496,5.749,148.568
C04972=1214.147,108.637,-49.392,-178.494,5.750,148.567
C04973=1214.143,108.887,-49.411,-178.491,5.752,148.567
C04974=1214.138,109.136,-49.429,-178.489,5.753,148.566
C04975=1214.133,109.385,-49.449,-178.486,5.753,148.566
C04976=1214.128,109.634,-49.468,-178.483,5.755,148.565
C04977=1214.124,109.883,-49.487,-178.481,5.756,148.565
C04978=1214.118,110.132,-49.507,-178.478,5.756,148.564
C04979=1214.114,110.382,-49.525,-178.475,5.758,148.564
C04980=1214.109,110.631,-49.544,-178.473,5.759,148.563
C04981=1214.105,110.880,-49.563,-178.471,5.760,148.563
C04982=1214.099,111.129,-49.583,-178.467,5.761,148.562
C04983=1214.095,111.379,-49.602,-178.465,5.762,148.561
C04984=1214.091,111.628,-49.621,-178.463,5.763,148.561
C04985=1214.085,111.877,-49.641,-178.460,5.764,148.560
C04986=1214.081,112.126,-49.660,-178.457,5.765,148.560
C04987=1214.076,112.376,-49.678,-178.455,5.766,148.559
C04988=1214.071,112.625,-49.698,-178.452,5.767,148.559
C04989=1214.066,112.874,-49.717,-178.450,5.768,148.558
C04990=1214.061,113.124,-49.737,-178.447,5.769,148.558
C04991=1214.056,113.372,-49.756,-178.444,5.770,148.557
C04992=1214.051,113.622,-49.775,-178.442,5.771,148.557
C04993=1214.047,113.871,-49.795,-178.439,5.772,148.556
C04994=1214.042,114.120,-49.814,-178.437,5.774,148.556
C04995=1214.037,114.369,-49.833,-178.434,5.774,148.555
C04996=1214.032,114.618,-49.853,-178.432,5.776,148.555
C04997=1214.027,114.868,-49.872,-178.429,5.777,148.554
C04998=1214.023,115.116,-49.891,-178.427,5.778,148.554
C04999=1214.018,115.366,-49.911,-178.424,5.779,148.553
C05000=1214.013,115.616,-49.930,-178.421,5.780,148.553
C05001=1214.008,115.864,-49.950,-178.419,5.781,148.552
C05002=1214.004,116.114,-49.969,-178.416,5.782,148.551
C05003=1213.998,116.362,-49.988,-178.414,5.783,148.551
C05004=1213.994,116.612,-50.008,-178.411,5.784,148.550
C05005=1213.989,116.862,-50.027,-178.408,5.785,148.550
C05006=1213.984,117.111,-50.046,-178.406,5.786,148.549
C05007=1213.980,117.360,-50.066,-178.403,5.788,148.549
C05008=1213.975,117.609,-50.086,-178.401,5.789,148.548
C05009=1213.970,117.858,-50.105,-178.398,5.789,148.548
C05010=1213.965,118.107,-50.125,-178.396,5.791,148.547
C05011=1213.960,118.357,-50.144,-178.393,5.792,148.547
C05012=1213.955,118.606,-50.164,-178.390,5.794,148.546
C05013=1213.951,118.855,-50.183,-178.388,5.794,148.546
C05014=1213.946,119.104,-50.203,-178.386,5.795,148.545
C05015=1213.941,119.353,-50.223,-178.382,5.797,148.545
C05016=1213.936,119.602,-50.242,-178.380,5.798,148.544
C05017=1213.932,119.852,-50.262,-178.378,5.798,148.544
C05018=1213.926,120.101,-50.281,-178.375,5.800,148.543
C05019=1213.922,120.350,-50.301,-178.372,5.801,148.543
C05020=1213.917,120.599,-50.321,-178.370,5.802,148.542
C05021=1213.913,120.848,-50.340,-178.367,5.803,148.542
C05022=1213.908,121.097,-50.359,-178.365,5.804,148.541
C05023=1213.903,121.347,-50.379,-178.362,5.805,148.540
C05024=1213.898,121.596,-50.398,-178.360,5.806,148.540
C05025=1213.893,121.845,-50.419,-178.356,5.808,148.539
C05026=1213.889,122.094,-50.438,-178.354,5.809,148.539
C05027=1213.884,122.344,-50.458,-178.352,5.809,148.538
C05028=1213.879,122.592,-50.478,-178.349,5.811,148.538
C05029=1213.874,122.842,-50.498,-178.346,5.812,148.537
C05030=1213.869,123.091,-50.517,-178.344,5.813,148.537
C05031=1213.864,123.339,-50.537,-178.341,5.814,148.536
C05032=1213.860,123.589,-50.557,-178.338,5.816,148.536
C05033=1213.855,123.839,-50.577,-178.336,5.816,148.535
C05034=1213.850,124.088,-50.597,-178.334,5.817,148.535
C05035=1213.845,124.336,-50.616,-178.331,5.819,148.534
C05036=1213.840,124.586,-50.636,-178.328,5.820,148.534
C05037=1213.836,124.835,-50.656,-178.326,5.822,148.533
C05038=1213.831,125.084,-50.676,-178.323,5.822,148.533
C05039=1213.826,125.333,-50.695,-178.321,5.823,148.532
C05040=1213.821,125.582,-50.716,-178.318,5.825,148.532
C05041=1213.817,125.832,-50.735,-178.316,5.826,148.531
C05042=1213.812,126.081,-50.756,-178.313,5.827,148.531
C05043=1213.807,126.330,-50.775,-178.310,5.828,148.530
C05044=1213.802,126.579,-50.795,-178.307,5.829,148.530
C05045=1213.798,126.828,-50.815,-178.305,5.830,148.529
C05046=1213.793,127.078,-50.835,-178.302,5.832,148.529
C05047=1213.788,127.327,-50.855,-178.300,5.833,148.528
C05048=1213.784,127.576,-50.875,-178.297,5.833,148.528
C05049=1213.779,127.825,-50.895,-178.295,5.835,148.527
C05050=1213.774,128.074,-50.914,-178.292,5.836,148.527
C05051=1213.769,128.323,-50.935,-178.289,5.838,148.526
C05052=1213.765,128.573,-50.954,-178.287,5.839,148.526
C05053=1213.760,128.822,-50.975,-178.284,5.840,148.525
C05054=1213.755,129.071,-50.996,-178.282,5.841,148.525
C05055=1213.750,129.320,-51.015,-178.279,5.842,148.524
C05056=1213.745,129.569,-51.035,-178.277,5.843,148.524
C05057=1213.741,129.818,-51.055,-178.274,5.844,148.523
C05058=1213.736,130.067,-51.076,-178.271,5.846,148.523
C05059=1213.731,130.317,-51.095,-178.269,5.847,148.522
C05060=1213.727,130.566,-51.116,-178.266,5.848,148.522
C05061=1213.721,130.814,-51.136,-178.264,5.849,148.521
C05062=1213.716,131.064,-51.156,-178.261,5.851,148.521
C05063=1213.712,131.313,-51.176,-178.259,5.852,148.520
C05064=1213.708,131.562,-51.197,-178.255,5.853,148.520
C05065=1213.703,131.811,-51.216,-178.253,5.854,148.519
C05066=1213.698,132.061,-51.237,-178.251,5.856,148.519
C05067=1213.693,132.310,-51.257,-178.248,5.856,148.518
C05068=1213.688,132.559,-51.277,-178.246,5.857,148.518
C05069=1213.683,132.807,-51.297,-178.243,5.859,148.517
C05070=1213.678,133.077,-51.319,-178.240,5.861,148.517
C05071=1213.674,133.345,-51.341,-178.237,5.861,148.516
C05072=1213.668,133.614,-51.363,-178.234,5.863,148.516
C05073=1213.663,133.882,-51.385,-178.232,5.864,148.515
C05074=1213.658,134.131,-51.406,-178.229,5.865,148.515
C05075=1213.654,134.381,-51.425,-178.226,5.867,148.514
C05076=1213.649,134.630,-51.446,-178.224,5.868,148.514
C05077=1213.644,134.879,-51.467,-178.221,5.869,148.513
C05078=1213.640,135.128,-51.487,-178.219,5.870,148.513
C05079=1213.635,135.378,-51.507,-178.216,5.872,148.512
C05080=1213.630,135.627,-51.527,-178.214,5.873,148.512
C05081=1213.625,135.876,-51.548,-178.211,5.874,148.511
C05082=1213.620,136.124,-51.568,-178.208,5.875,148.511
C05083=1213.616,136.373,-51.588,-178.206,5.877,148.510
C05084=1213.610,136.623,-51.608,-178.203,5.877,148.510
C05085=1213.606,136.872,-51.629,-178.200,5.879,148.509
C05086=1213.601,137.121,-51.649,-178.198,5.880,148.509
C05087=1213.596,137.370,-51.670,-178.195,5.882,148.508
C05088=1213.592,137.619,-51.691,-178.193,5.883,148.508
C05089=1213.587,137.868,-51.711,-178.190,5.884,148.507
C05090=1213.582,138.117,-51.732,-178.188,5.885,148.507
C05091=1213.578,138.366,-51.752,-178.185,5.887,148.507
C05092=1213.572,138.616,-51.773,-178.182,5.887,148.506
C05093=1213.568,138.865,-51.793,-178.180,5.889,148.506
C05094=1213.563,139.114,-51.813,-178.177,5.890,148.505
C05095=1213.558,139.363,-51.834,-178.175,5.892,148.505
C05096=1213.554,139.612,-51.855,-178.172,5.893,148.504
C05097=1213.549,139.861,-51.875,-178.169,5.894,148.504
C05098=1213.544,140.110,-51.896,-178.167,5.895,148.503
C05099=1213.540,140.359,-51.916,-178.164,5.897,148.503
C05100=1213.535,140.608,-51.937,-178.162,5.897,148.502
C05101=1213.530,140.857,-51.958,-178.159,5.899,148.502
C05102=1213.525,141.107,-51.979,-178.157,5.900,148.501
C05103=1213.520,141.356,-51.999,-178.154,5.902,148.501
C05104=1213.516,141.605,-52.019,-178.152,5.903,148.500
C05105=1213.511,141.854,-52.040,-178.149,5.904,148.500
C05106=1213.507,142.104,-52.061,-178.147,5.905,148.499
C05107=1213.502,142.353,-52.082,-178.144,5.907,148.499
C05108=1213.497,142.602,-52.102,-178.141,5.907,148.498
C05109=1213.493,142.850,-52.124,-178.139,5.909,148.498
C05110=1213.488,143.099,-52.144,-178.136,5.910,148.497
C05111=1213.483,143.349,-52.165,-178.133,5.912,148.497
C05112=1213.479,143.598,-52.186,-178.131,5.913,148.497
C05113=1213.473,143.847,-52.207,-178.128,5.914,148.496
C05114=1213.469,144.096,-52.227,-178.125,5.916,148.496
C05115=1213.464,144.345,-52.248,-178.123,5.917,148.495
C05116=1213.459,144.594,-52.268,-178.120,5.918,148.495
C05117=1213.454,144.843,-52.290,-178.118,5.919,148.494
C05118=1213.451,145.092,-52.311,-178.115,5.921,148.494
C05119=1213.445,145.341,-52.332,-178.113,5.922,148.493
C05120=1213.440,145.591,-52.353,-178.110,5.924,148.493
C05121=1213.436,145.840,-52.373,-178.108,5.925,148.492
C05122=1213.431,146.088,-52.395,-178.105,5.926,148.492
C05123=1213.426,146.337,-52.415,-178.102,5.928,148.491
C05124=1213.421,146.587,-52.436,-178.100,5.928,148.491
C05125=1213.417,146.835,-52.457,-178.097,5.930,148.490
C05126=1213.412,147.085,-52.478,-178.095,5.931,148.490
C05127=1213.407,147.334,-52.500,-178.092,5.933,148.489
C05128=1213.403,147.583,-52.520,-178.089,5.934,148.489
C05129=1213.398,147.832,-52.541,-178.087,5.935,148.489
C05130=1213.394,148.081,-52.562,-178.084,5.936,148.488
C05131=1213.389,148.330,-52.583,-178.082,5.938,148.488
C05132=1213.383,148.579,-52.604,-178.079,5.940,148.487
C05133=1213.379,148.829,-52.625,-178.076,5.940,148.487
C05134=1213.375,149.077,-52.646,-178.074,5.942,148.486
C05135=1213.369,149.327,-52.667,-178.071,5.943,148.486
C05136=1213.365,149.576,-52.688,-178.068,5.945,148.485
C05137=1213.360,149.824,-52.709,-178.066,5.945,148.485
C05138=1213.356,150.074,-52.731,-178.064,5.947,148.485
C05139=1213.351,150.323,-52.752,-178.061,5.949,148.484
C05140=1213.346,150.572,-52.773,-178.058,5.950,148.484
C05141=1213.341,150.821,-52.794,-178.056,5.952,148.483
C05142=1213.337,151.069,-52.815,-178.053,5.952,148.483
C05143=1213.332,151.319,-52.836,-178.050,5.954,148.482
C05144=1213.328,151.568,-52.858,-178.048,5.956,148.482
C05145=1213.322,151.817,-52.879,-178.046,5.957,148.481
C05146=1213.318,152.066,-52.900,-178.042,5.958,148.481
C05147=1213.313,152.315,-52.921,-178.040,5.959,148.480
C05148=1213.308,152.565,-52.942,-178.038,5.961,148.480
C05149=1213.304,152.813,-52.964,-178.035,5.962,148.479
C05150=1213.299,153.062,-52.984,-178.032,5.963,148.479
C05151=1213.294,153.311,-53.006,-178.030,5.965,148.479
C05152=1213.290,153.561,-53.027,-178.028,5.966,148.478
C05153=1213.285,153.810,-53.049,-178.024,5.968,148.478
C05154=1213.280,154.059,-53.070,-178.022,5.969,148.477
C05155=1213.276,154.307,-53.091,-178.020,5.970,148.477
C05156=1213.271,154.557,-53.113,-178.016,5.972,148.476
C05157=1213.266,154.806,-53.134,-178.014,5.973,148.476
C05158=1213.261,155.054,-53.156,-178.012,5.975,148.476
C05159=1213.256,155.304,-53.177,-178.009,5.976,148.475
C05160=1213.253,155.553,-53.198,-178.006,5.977,148.475
C05161=1213.247,155.802,-53.219,-178.004,5.979,148.474
C05162=1213.242,156.051,-53.241,-178.002,5.980,148.474
C05163=1213.238,156.300,-53.263,-177.999,5.981,148.473
C05164=1213.233,156.549,-53.284,-177.996,5.983,148.473
C05165=1213.228,156.798,-53.306,-177.994,5.984,148.472
C05166=1213.223,157.047,-53.327,-177.991,5.986,148.472
C05167=1213.219,157.296,-53.348,-177.988,5.987,148.471
C05168=1213.215,157.545,-53.370,-177.986,5.988,148.471
C05169=1213.210,157.793,-53.391,-177.983,5.990,148.471
C05170=1213.205,158.043,-53.413,-177.981,5.991,148.470
C05171=1213.200,158.292,-53.434,-177.978,5.993,148.470
C05172=1213.195,158.541,-53.456,-177.975,5.994,148.469
C05173=1213.191,158.791,-53.477,-177.973,5.995,148.469
C05174=1213.186,159.059,-53.501,-177.970,5.997,148.468
C05175=1213.181,159.328,-53.524,-177.967,5.999,148.468
C05176=1213.175,159.598,-53.548,-177.964,6.000,148.467
C05177=1213.171,159.866,-53.571,-177.961,6.002,148.467
C05178=1213.166,160.116,-53.592,-177.959,6.003,148.467
C05179=1213.161,160.364,-53.614,-177.956,6.004,148.466
C05180=1213.157,160.614,-53.636,-177.954,6.006,148.466
C05181=1213.152,160.862,-53.657,-177.951,6.007,148.465
C05182=1213.148,161.112,-53.679,-177.948,6.009,148.465
C05183=1213.142,161.361,-53.700,-177.946,6.011,148.464
C05184=1213.137,161.609,-53.722,-177.944,6.011,148.464
C05185=1213.133,161.859,-53.744,-177.941,6.013,148.464
C05186=1213.128,162.107,-53.766,-177.938,6.015,148.463
C05187=1213.124,162.357,-53.788,-177.936,6.016,148.463
C05188=1213.119,162.605,-53.810,-177.933,6.018,148.462
C05189=1213.114,162.854,-53.831,-177.931,6.019,148.462
C05190=1213.110,163.103,-53.853,-177.928,6.020,148.461
C05191=1213.105,163.353,-53.874,-177.925,6.022,148.461
C05192=1213.101,163.602,-53.896,-177.923,6.023,148.460
C05193=1213.096,163.851,-53.918,-177.920,6.025,148.460
C05194=1213.091,164.100,-53.940,-177.918,6.026,148.460
C05195=1213.087,164.349,-53.962,-177.915,6.027,148.459
C05196=1213.082,164.597,-53.983,-177.912,6.029,148.459
C05197=1213.077,164.847,-54.005,-177.910,6.031,148.458
C05198=1213.072,165.096,-54.028,-177.907,6.032,148.458
C05199=1213.068,165.345,-54.050,-177.904,6.033,148.457
C05200=1213.063,165.593,-54.071,-177.902,6.035,148.457
C05201=1213.058,165.843,-54.093,-177.899,6.037,148.457
C05202=1213.054,166.091,-54.115,-177.897,6.038,148.456
C05203=1213.049,166.341,-54.137,-177.894,6.039,148.456
C05204=1213.044,166.589,-54.159,-177.891,6.041,148.455
C05205=1213.040,166.839,-54.181,-177.889,6.042,148.455
C05206=1213.035,167.088,-54.203,-177.886,6.044,148.455
C05207=1213.030,167.337,-54.225,-177.884,6.046,148.454
C05208=1213.025,167.586,-54.247,-177.881,6.046,148.454
C05209=1213.022,167.834,-54.270,-177.879,6.048,148.453
C05210=1213.017,168.083,-54.291,-177.876,6.050,148.453
C05211=1213.012,168.332,-54.313,-177.874,6.051,148.452
C05212=1213.007,168.581,-54.336,-177.871,6.053,148.452
C05213=1213.002,168.831,-54.358,-177.868,6.054,148.452
C05214=1212.998,169.079,-54.379,-177.865,6.056,148.451
C05215=1212.993,169.329,-54.402,-177.863,6.057,148.451
C05216=1212.988,169.577,-54.423,-177.861,6.059,148.450
C05217=1212.984,169.826,-54.447,-177.858,6.061,148.450
C05218=1212.979,170.075,-54.468,-177.855,6.061,148.449
C05219=1212.975,170.324,-54.490,-177.853,6.063,148.449
C05220=1212.970,170.573,-54.512,-177.850,6.065,148.449
C05221=1212.965,170.823,-54.535,-177.848,6.066,148.448
C05222=1212.960,171.071,-54.557,-177.845,6.068,148.448
C05223=1212.956,171.320,-54.579,-177.842,6.069,148.447
C05224=1212.951,171.569,-54.601,-177.839,6.071,148.447
C05225=1212.946,171.818,-54.623,-177.837,6.072,148.447
C05226=1212.942,172.067,-54.646,-177.835,6.074,148.446
C05227=1212.937,172.316,-54.668,-177.832,6.076,148.446
C05228=1212.932,172.565,-54.690,-177.829,6.077,148.445
C05229=1212.928,172.813,-54.713,-177.827,6.078,148.445
C05230=1212.923,173.063,-54.735,-177.824,6.080,148.445
C05231=1212.918,173.312,-54.758,-177.821,6.082,148.444
C05232=1212.914,173.561,-54.779,-177.819,6.083,148.444
C05233=1212.910,173.810,-54.802,-177.817,6.085,148.443
C05234=1212.904,174.059,-54.824,-177.813,6.086,148.443
C05235=1212.900,174.307,-54.847,-177.811,6.088,148.443
C05236=1212.896,174.557,-54.869,-177.809,6.089,148.442
C05237=1212.890,174.806,-54.891,-177.806,6.091,148.442
C05238=1212.886,175.054,-54.914,-177.803,6.092,148.441
C05239=1212.881,175.303,-54.936,-177.801,6.094,148.441
C05240=1212.876,175.553,-54.958,-177.798,6.095,148.440
C05241=1212.872,175.801,-54.981,-177.796,6.097,148.440
C05242=1212.867,176.050,-55.004,-177.793,6.099,148.440
C05243=1212.863,176.299,-55.026,-177.790,6.100,148.439
C05244=1212.858,176.548,-55.048,-177.788,6.101,148.439
C05245=1212.853,176.797,-55.071,-177.785,6.103,148.439
C05246=1212.849,177.046,-55.093,-177.782,6.105,148.438
C05247=1212.844,177.295,-55.117,-177.780,6.106,148.438
C05248=1212.839,177.544,-55.138,-177.778,6.107,148.437
C05249=1212.835,177.793,-55.162,-177.775,6.109,148.437
C05250=1212.830,178.042,-55.184,-177.772,6.111,148.437
C05251=1212.826,178.290,-55.206,-177.770,6.113,148.436
C05252=1212.821,178.540,-55.229,-177.767,6.114,148.436
C05253=1212.817,178.789,-55.252,-177.764,6.115,148.435
C05254=1212.811,179.037,-55.274,-177.762,6.117,148.435
C05255=1212.807,179.286,-55.297,-177.759,6.119,148.435
C05256=1212.803,179.535,-55.320,-177.757,6.120,148.434
C05257=1212.798,179.784,-55.342,-177.754,6.122,148.434
C05258=1212.793,180.033,-55.365,-177.752,6.124,148.433
C05259=1212.789,180.282,-55.387,-177.749,6.125,148.433
C05260=1212.784,180.531,-55.410,-177.746,6.127,148.433
C05261=1212.779,180.779,-55.433,-177.744,6.128,148.432
C05262=1212.774,181.029,-55.455,-177.741,6.130,148.432
C05263=1212.770,181.278,-55.479,-177.738,6.132,148.431
C05264=1212.766,181.527,-55.502,-177.736,6.133,148.431
C05265=1212.760,181.776,-55.524,-177.734,6.134,148.431
C05266=1212.756,182.024,-55.547,-177.731,6.136,148.430
C05267=1212.752,182.273,-55.570,-177.728,6.138,148.430
C05268=1212.747,182.523,-55.592,-177.725,6.140,148.429
C05269=1212.742,182.771,-55.615,-177.723,6.141,148.429
C05270=1212.737,183.020,-55.638,-177.720,6.142,148.429
C05271=1212.733,183.269,-55.660,-177.718,6.144,148.428
C05272=1212.728,183.518,-55.684,-177.715,6.146,148.428
C05273=1212.724,183.766,-55.706,-177.713,6.148,148.428
C05274=1212.719,184.016,-55.730,-177.710,6.150,148.427
C05275=1212.714,184.265,-55.753,-177.708,6.151,148.427
C05276=1212.710,184.514,-55.775,-177.705,6.152,148.427
C05277=1212.705,184.763,-55.798,-177.702,6.154,148.426
C05278=1212.700,185.033,-55.823,-177.699,6.156,148.426
C05279=1212.695,185.302,-55.848,-177.697,6.158,148.425
C05280=1212.690,185.572,-55.873,-177.694,6.159,148.425
C05281=1212.686,185.841,-55.897,-177.691,6.161,148.424
C05282=1212.681,186.090,-55.921,-177.688,6.163,148.424
C05283=1212.676,186.339,-55.944,-177.686,6.165,148.424
C05284=1212.671,186.588,-55.967,-177.683,6.166,148.423
C05285=1212.667,186.836,-55.990,-177.681,6.167,148.423
C05286=1212.662,187.086,-56.013,-177.678,6.169,148.423
C05287=1212.658,187.335,-56.036,-177.676,6.171,148.422
C05288=1212.654,187.583,-56.059,-177.673,6.173,148.422
C05289=1212.648,187.832,-56.082,-177.670,6.175,148.421
C05290=1212.644,188.081,-56.106,-177.668,6.176,148.421
C05291=1212.639,188.330,-56.128,-177.665,6.177,148.421
C05292=1212.635,188.579,-56.151,-177.662,6.179,148.420
C05293=1212.630,188.828,-56.174,-177.660,6.181,148.420
C05294=1212.625,189.077,-56.198,-177.657,6.183,148.419
C05295=1212.620,189.326,-56.221,-177.654,6.184,148.419
C05296=1212.616,189.574,-56.243,-177.652,6.185,148.419
C05297=1212.611,189.823,-56.267,-177.650,6.187,148.418
C05298=1212.607,190.072,-56.290,-177.647,6.189,148.418
C05299=1212.602,190.321,-56.314,-177.644,6.191,148.418
C05300=1212.597,190.570,-56.337,-177.642,6.193,148.417
C05301=1212.593,190.819,-56.361,-177.639,6.195,148.417
C05302=1212.589,191.067,-56.384,-177.637,6.196,148.417
C05303=1212.584,191.316,-56.407,-177.634,6.197,148.416
C05304=1212.579,191.565,-56.430,-177.632,6.199,148.416
C05305=1212.575,191.814,-56.454,-177.629,6.201,148.416
C05306=1212.570,192.064,-56.477,-177.626,6.203,148.415
C05307=1212.565,192.312,-56.500,-177.623,6.204,148.415
C05308=1212.561,192.561,-56.523,-177.621,6.206,148.414
C05309=1212.556,192.810,-56.546,-177.618,6.207,148.414
C05310=1212.552,193.058,-56.570,-177.616,6.209,148.414
C05311=1212.547,193.307,-56.594,-177.613,6.211,148.413
C05312=1212.542,193.556,-56.617,-177.611,6.213,148.413
C05313=1212.538,193.805,-56.640,-177.608,6.215,148.413
C05314=1212.533,194.054,-56.664,-177.605,6.216,148.412
C05315=1212.528,194.303,-56.687,-177.603,6.218,148.412
C05316=1212.524,194.552,-56.711,-177.600,6.219,148.411
C05317=1212.519,194.801,-56.735,-177.598,6.221,148.411
C05318=1212.514,195.050,-56.758,-177.595,6.223,148.411
C05319=1212.510,195.299,-56.781,-177.593,6.225,148.410
C05320=1212.505,195.547,-56.805,-177.590,6.227,148.410
C05321=1212.501,195.796,-56.828,-177.587,6.228,148.410
C05322=1212.497,196.045,-56.852,-177.585,6.230,148.409
C05323=1212.492,196.294,-56.875,-177.582,6.232,148.409
C05324=1212.487,196.542,-56.899,-177.579,6.234,148.409
C05325=1212.483,196.791,-56.922,-177.577,6.235,148.408
C05326=1212.478,197.040,-56.946,-177.575,6.237,148.408
C05327=1212.474,197.289,-56.970,-177.572,6.238,148.408
C05328=1212.469,197.538,-56.993,-177.569,6.240,148.407
C05329=1212.464,197.787,-57.016,-177.567,6.242,148.407
C05330=1212.460,198.035,-57.041,-177.564,6.244,148.407
C05331=1212.454,198.285,-57.065,-177.561,6.246,148.406
C05332=1212.450,198.533,-57.089,-177.559,6.248,148.406
C05333=1212.445,198.782,-57.112,-177.556,6.249,148.406
C05334=1212.441,199.031,-57.135,-177.554,6.250,148.405
C05335=1212.436,199.279,-57.159,-177.551,6.252,148.405
C05336=1212.432,199.529,-57.183,-177.548,6.254,148.404
C05337=1212.427,199.777,-57.207,-177.546,6.256,148.404
C05338=1212.422,200.026,-57.230,-177.543,6.257,148.404
C05339=1212.419,200.275,-57.255,-177.540,6.259,148.403
C05340=1212.414,200.524,-57.278,-177.538,6.261,148.403
C05341=1212.410,200.773,-57.302,-177.535,6.263,148.403
C05342=1212.405,201.022,-57.325,-177.532,6.265,148.402
C05343=1212.400,201.270,-57.349,-177.530,6.267,148.402
C05344=1212.395,201.519,-57.373,-177.528,6.268,148.402
C05345=1212.391,201.768,-57.397,-177.525,6.269,148.401
C05346=1212.386,202.017,-57.421,-177.522,6.271,148.401
C05347=1212.382,202.265,-57.445,-177.520,6.273,148.401
C05348=1212.377,202.514,-57.468,-177.517,6.275,148.400
C05349=1212.373,202.763,-57.493,-177.515,6.277,148.400
C05350=1212.368,203.013,-57.517,-177.512,6.279,148.400
C05351=1212.363,203.261,-57.541,-177.510,6.281,148.399
C05352=1212.359,203.509,-57.565,-177.507,6.283,148.399
C05353=1212.354,203.759,-57.588,-177.504,6.284,148.399
C05354=1212.350,204.007,-57.612,-177.502,6.286,148.398
C05355=1212.345,204.255,-57.636,-177.499,6.288,148.398
C05356=1212.341,204.505,-57.661,-177.496,6.290,148.398
C05357=1212.336,204.754,-57.685,-177.494,6.292,148.397
C05358=1212.332,205.002,-57.709,-177.492,6.293,148.397
C05359=1212.327,205.251,-57.732,-177.489,6.295,148.397
C05360=1212.322,205.500,-57.757,-177.486,6.296,148.396
C05361=1212.317,205.748,-57.781,-177.484,6.298,148.396
C05362=1212.313,205.998,-57.805,-177.481,6.300,148.396
C05363=1212.309,206.247,-57.829,-177.478,6.302,148.395
C05364=1212.304,206.495,-57.853,-177.476,6.304,148.395
C05365=1212.299,206.744,-57.877,-177.473,6.306,148.395
C05366=1212.295,206.993,-57.901,-177.470,6.308,148.394
C05367=1212.290,207.242,-57.926,-177.468,6.309,148.394
C05368=1212.286,207.491,-57.950,-177.465,6.311,148.394
C05369=1212.281,207.739,-57.974,-177.463,6.313,148.393
C05370=1212.276,207.988,-57.998,-177.460,6.315,148.393
C05371=1212.272,208.237,-58.022,-177.457,6.317,148.393
C05372=1212.268,208.486,-58.046,-177.455,6.319,148.392
C05373=1212.263,208.735,-58.071,-177.452,6.320,148.392
C05374=1212.258,208.983,-58.095,-177.449,6.322,148.392
C05375=1212.254,209.231,-58.119,-177.447,6.324,148.391
C05376=1212.249,209.481,-58.144,-177.444,6.326,148.391
C05377=1212.245,209.730,-58.168,-177.442,6.328,148.391
C05378=1212.240,209.978,-58.192,-177.439,6.330,148.390
C05379=1212.235,210.227,-58.216,-177.437,6.332,148.390
C05380=1212.231,210.476,-58.241,-177.434,6.334,148.390
C05381=1212.226,210.725,-58.266,-177.431,6.335,148.389
C05382=1212.222,210.995,-58.292,-177.429,6.337,148.389
C05383=1212.216,211.265,-58.318,-177.426,6.339,148.389
C05384=1212.211,211.536,-58.344,-177.423,6.341,148.388
C05385=1212.207,211.806,-58.371,-177.420,6.342,148.388
C05386=1212.202,212.055,-58.396,-177.418,6.344,148.387
C05387=1212.197,212.304,-58.420,-177.415,6.346,148.387
C05388=1212.193,212.553,-58.445,-177.413,6.348,148.387
C05389=1212.188,212.801,-58.469,-177.410,6.350,148.387
C05390=1212.184,213.050,-58.493,-177.408,6.352,148.386
C05391=1212.179,213.299,-58.518,-177.405,6.354,148.386
C05392=1212.175,213.548,-58.542,-177.402,6.356,148.386
C05393=1212.170,213.796,-58.567,-177.400,6.357,148.385
C05394=1212.165,214.045,-58.591,-177.397,6.359,148.385
C05395=1212.161,214.294,-58.616,-177.394,6.361,148.385
C05396=1212.156,214.543,-58.640,-177.392,6.363,148.384
C05397=1212.152,214.791,-58.666,-177.389,6.365,148.384
C05398=1212.148,215.040,-58.690,-177.386,6.367,148.384
C05399=1212.143,215.289,-58.715,-177.384,6.369,148.384
C05400=1212.138,215.537,-58.739,-177.382,6.371,148.383
C05401=1212.134,215.786,-58.764,-177.379,6.373,148.383
C05402=1212.129,216.035,-58.788,-177.376,6.374,148.383
C05403=1212.125,216.284,-58.813,-177.374,6.376,148.382
C05404=1212.121,216.532,-58.838,-177.371,6.378,148.382
C05405=1212.116,216.781,-58.863,-177.368,6.381,148.382
C05406=1212.111,217.030,-58.888,-177.365,6.383,148.381
C05407=1212.107,217.279,-58.912,-177.363,6.384,148.381
C05408=1212.102,217.527,-58.936,-177.360,6.387,148.381
C05409=1212.098,217.776,-58.961,-177.358,6.388,148.381
C05410=1212.093,218.025,-58.986,-177.355,6.390,148.380
C05411=1212.088,218.274,-59.011,-177.353,6.392,148.380
C05412=1212.084,218.522,-59.035,-177.350,6.394,148.380
C05413=1212.079,218.771,-59.061,-177.347,6.396,148.379
C05414=1212.075,219.020,-59.086,-177.345,6.398,148.379
C05415=1212.070,219.268,-59.110,-177.342,6.400,148.379
C05416=1212.066,219.517,-59.135,-177.339,6.401,148.378
C05417=1212.062,219.766,-59.160,-177.337,6.404,148.378
C05418=1212.057,220.015,-59.185,-177.335,6.405,148.378
C05419=1212.052,220.263,-59.210,-177.332,6.407,148.377
C05420=1212.047,220.512,-59.235,-177.329,6.409,148.377
C05421=1212.043,220.761,-59.259,-177.327,6.411,148.377
C05422=1212.039,221.009,-59.284,-177.324,6.413,148.376
C05423=1212.034,221.258,-59.309,-177.321,6.415,148.376
C05424=1212.030,221.506,-59.334,-177.319,6.417,148.376
C05425=1212.025,221.756,-59.359,-177.317,6.419,148.376
C05426=1212.020,222.004,-59.384,-177.314,6.420,148.375
C05427=1212.016,222.253,-59.410,-177.311,6.422,148.375
C05428=1212.012,222.502,-59.434,-177.309,6.424,148.375
C05429=1212.007,222.750,-59.460,-177.306,6.426,148.374
C05430=1212.002,222.999,-59.484,-177.304,6.428,148.374
C05431=1211.998,223.248,-59.510,-177.301,6.430,148.374
C05432=1211.994,223.496,-59.534,-177.299,6.432,148.374
C05433=1211.989,223.745,-59.560,-177.296,6.434,148.373
C05434=1211.984,223.994,-59.584,-177.293,6.436,148.373
C05435=1211.980,224.243,-59.610,-177.291,6.437,148.373
C05436=1211.975,224.491,-59.635,-177.289,6.440,148.373
C05437=1211.971,224.740,-59.660,-177.285,6.442,148.372
C05438=1211.966,224.989,-59.685,-177.283,6.444,148.372
C05439=1211.962,225.237,-59.710,-177.280,6.446,148.372
C05440=1211.957,225.486,-59.736,-177.277,6.448,148.371
C05441=1211.953,225.735,-59.761,-177.275,6.450,148.371
C05442=1211.948,225.983,-59.786,-177.273,6.452,148.371
C05443=1211.944,226.232,-59.811,-177.270,6.454,148.371
C05444=1211.940,226.481,-59.836,-177.267,6.456,148.370
C05445=1211.935,226.729,-59.862,-177.265,6.457,148.370
C05446=1211.931,226.979,-59.887,-177.262,6.459,148.370
C05447=1211.926,227.227,-59.912,-177.260,6.461,148.369
C05448=1211.921,227.475,-59.938,-177.257,6.463,148.369
C05449=1211.916,227.724,-59.963,-177.255,6.465,148.369
C05450=1211.912,227.973,-59.988,-177.252,6.467,148.368
C05451=1211.908,228.222,-60.014,-177.249,6.469,148.368
C05452=1211.903,228.470,-60.039,-177.247,6.471,148.368
C05453=1211.899,228.719,-60.064,-177.245,6.473,148.368
C05454=1211.894,228.967,-60.089,-177.242,6.475,148.367
C05455=1211.890,229.216,-60.115,-177.239,6.477,148.367
C05456=1211.886,229.465,-60.140,-177.236,6.479,148.367
C05457=1211.881,229.713,-60.166,-177.234,6.481,148.367
C05458=1211.877,229.962,-60.191,-177.231,6.483,148.366
C05459=1211.872,230.210,-60.217,-177.229,6.485,148.366
C05460=1211.867,230.460,-60.242,-177.226,6.487,148.366
C05461=1211.863,230.709,-60.267,-177.224,6.489,148.366
C05462=1211.858,230.957,-60.293,-177.221,6.491,148.365
C05463=1211.854,231.205,-60.319,-177.219,6.493,148.365
C05464=1211.850,231.454,-60.344,-177.216,6.495,148.365
C05465=1211.845,231.702,-60.370,-177.214,6.496,148.364
C05466=1211.841,231.951,-60.396,-177.211,6.499,148.364
C05467=1211.836,232.201,-60.421,-177.208,6.501,148.364
C05468=1211.831,232.449,-60.446,-177.206,6.503,148.364
C05469=1211.827,232.698,-60.472,-177.203,6.505,148.363
C05470=1211.823,232.946,-60.497,-177.201,6.507,148.363
C05471=1211.817,233.195,-60.523,-177.198,6.509,148.363
C05472=1211.813,233.444,-60.549,-177.196,6.511,148.363
C05473=1211.809,233.692,-60.575,-177.193,6.513,148.362
C05474=1211.804,233.940,-60.600,-177.191,6.515,148.362
C05475=1211.800,234.189,-60.626,-177.188,6.517,148.362
C05476=1211.796,234.438,-60.652,-177.186,6.519,148.361
C05477=1211.791,234.686,-60.677,-177.182,6.521,148.361
C05478=1211.787,234.935,-60.703,-177.180,6.524,148.361
C05479=1211.782,235.184,-60.729,-177.178,6.525,148.361
